// TwinCAT 3 PLC project XtsTransport
// Title: XTS Transport
// Author: HAUD
// ProjectVersion: 4.02.16
// Description: . XTS_TRANSPORT_LAYER by Daniel Hauer
// ProgramVersion: 3.1.4026.22
// libraries:
//   Tc2_EtherCAT, * (Beckhoff Automation GmbH)
//   Tc2_Math, * (Beckhoff Automation GmbH)
//   Tc2_MC2, * (Beckhoff Automation GmbH)
//   Tc2_Standard, * (Beckhoff Automation GmbH)
//   Tc2_System, * (Beckhoff Automation GmbH)
//   Tc2_Utilities, * (Beckhoff Automation GmbH)
//   Tc2_XmlDataSrv, * (Beckhoff Automation GmbH)
//   Tc3_McCollisionAvoidance, * (Beckhoff Automation GmbH)
//   Tc3_McCoordinatedMotion, * (Beckhoff Automation GmbH)
//   Tc3_Module, * (Beckhoff Automation GmbH)
//   Tc3_XTS_Utility, * (Beckhoff Automation GmbH)
//   VisuDialogs, * (System)
// project tree:
//   APPLICATION/ GVL_APPLICATION.TcGVL, MAIN_APP.TcPOU
//   APPLICATION/_config/ StationParameterExample.TcPOU
//   APPLICATION/_types/Application/ E_APP_CHECK.TcDUT, E_APP_VARIANT.TcDUT, ST_APP_CTRL.TcDUT, ST_APP_STATE.TcDUT
//   APPLICATION/_types/Collector/ E_PROCESS_CHECK.TcDUT, E_PROCESS_CTRL.TcDUT, E_PROCESS_STATE.TcDUT, fb_ProcessCollector.TcPOU, fb_StationCollector.TcPOU, I_ProcessCollector.TcIO, ST_PROCESS_CTRL.TcDUT, ST_PROCESS_STATE.TcDUT
//   APPLICATION/_types/ fb_ProcessConductor.TcPOU
//   APPLICATION/_types/Instance/ E_INSTANCE.TcDUT, E_INSTANCE_CHECK.TcDUT, E_INSTANCE_CMD.TcDUT, E_INSTANCE_STATE.TcDUT, fb_Instance.TcPOU, ST_INSTANCE_CTRL.TcDUT, ST_INSTANCE_STATE.TcDUT
//   APPLICATION/_types/LinkedList/ E_LIST_CHECK.TcDUT, E_LIST_CTRL.TcDUT, E_LIST_STATE.TcDUT, fb_Process_LinkedList.TcPOU, fb_Process_LinkedListCtrl.TcPOU, I_Process_LinkedList.TcIO, ST_LIST_CTRL.TcDUT, ST_LIST_NODE_DATA.TcDUT, ST_LIST_STATE.TcDUT, ST_PROCESS_DATA.TcDUT, ST_PROCESS_LIST_RESULT.TcDUT
//   / GlobalTextList.TcGTLO, PlcTask.TcTTO
//   MAPPING/ MAPPING_XTS_in.TcPOU, MAPPING_XTS_out.TcPOU
//   MAPPING/_types/ E_MAPPING_CHECK.TcDUT, U_APP_CTRL.TcDUT, U_APP_STATE.TcDUT, U_GEAR_DATA.TcDUT, U_INSTANCE_CTRL.TcDUT, U_INSTANCE_STATE.TcDUT, U_MOVER_CTRL.TcDUT, U_MOVER_INFO.TcDUT, U_MOVER_SELECTOR_CTRL.TcDUT, U_MOVER_SELECTOR_STATE.TcDUT, U_MOVER_STATE.TcDUT, U_MOVE_DATA.TcDUT, U_TICKET_LIST_CTRL.TcDUT, U_TICKET_LIST_DATA_INPUT.TcDUT, U_TICKET_LIST_DATA_OUTPUT.TcDUT, U_TICKET_LIST_STATE.TcDUT, U_XTS_STATION_CTRL.TcDUT, U_XTS_STATION_STATE.TcDUT, U_XTS_TRANSPORT_CTRL.TcDUT, U_XTS_TRANSPORT_STATE.TcDUT
//   _MSG/class/ fb_LocalTime.TcPOU, fb_MessageData.TcPOU, fb_MessageDataCtrl.TcPOU
//   _MSG/ f_MessageSet.TcPOU, GVL_MSG_AXIS.TcGVL, GVL_MSG_XTS.TcGVL, I_MessageData.TcIO
//   _MSG/types/ e_Device.TcDUT, E_MessageType.TcDUT, E_MESSAGE_BATCH.TcDUT (not stored), E_MESSAGE_CHECK.TcDUT, E_MESSAGE_CTRL.TcDUT, E_MESSAGE_FLOW.TcDUT, E_MESSAGE_STATE.TcDUT, e_Subdevice.TcDUT, ST_Message.TcDUT, ST_MESSAGE_CTRL.TcDUT, ST_MESSAGE_STATE.TcDUT (not stored), TL_E_MESSAGETYPE.TcTLO
//   PLC_MOTION/_GVL/ PLC_CONSTANT.TcGVL
//   _types/ E_CHECK_STATE.TcDUT, E_PROGRESS.TcDUT, f_GetProgress.TcPOU, f_GetState.TcPOU, T_PROCESS.TcDUT
//   _XML/Configuration/ fb_Configuration.TcPOU, I_Configuration_Station.TcIO
//   _XML/Configuration/types/ ST_Configuration.TcDUT
//   _XML/ fb_XmlBase.TcPOU (not stored)
//   _XML/PositionOffsets/ fb_MoverPositionOffsetData.TcPOU
//   _XML/PositionOffsets/types/ ST_MOVER_OFFSETS.TcDUT
//   _XML/types/ E_DATA_CHECK.TcDUT (not stored), E_DATA_CTRL.TcDUT (not stored), E_DATA_STATE.TcDUT, fb_XmlRead.TcPOU (not stored), fb_XmlWrite.TcPOU, ST_DATA_CTRL.TcDUT (not stored), ST_DATA_STATE.TcDUT
//   XTS_TRANSPORT/CaGroup/ FB_CaGroup.TcPOU, I_XtsTransport_CaGroup.TcIO
//   XTS_TRANSPORT/CaGroup/types/ E_CA_GROUP_STATE.TcDUT, E_GROUP_CHECK.TcDUT, ST_GROUP_INFO.TcDUT
//   XTS_TRANSPORT/ GVL_XTS.TcGVL, GVL_XTS_CONSTANTS.TcGVL (not stored), GVL_XTS_VERSION.TcGVL, MAIN_XTS.TcPOU
//   XTS_TRANSPORT/Mover/ fb_Mover.TcPOU, fb_MoverCtrl.TcPOU, fb_MoverSelector.TcPOU (not stored), I_XtsTransport_Mover.TcIO
//   XTS_TRANSPORT/Mover/types/ E_MOVER_CHECK.TcDUT (not stored), E_MOVER_CTRL.TcDUT, E_MOVER_SELECTOR.TcDUT (not stored), E_MOVER_STATE.TcDUT, ST_GEAR_DATA.TcDUT, ST_MOVER_CTRL.TcDUT, ST_MOVER_INFO.TcDUT, ST_MOVER_SELECTOR_CTRL.TcDUT (not stored), ST_MOVER_SELECTOR_STATE.TcDUT, ST_MOVER_STATE.TcDUT, ST_MOVE_DATA.TcDUT
//   XTS_TRANSPORT/Xpu/ I_XtsTransport_Xpu.TcIO, fb_Xpu.TcPOU, fb_XpuCtrl.TcPOU
//   XTS_TRANSPORT/XtsStation/ fb_StationGearInPos.TcPOU, fb_StationProcess.TcPOU, I_XtsTransport_Station.TcIO
//   XTS_TRANSPORT/XtsStation/types/ E_STATION_CHECK.TcDUT, E_STATION_CTRL.TcDUT, E_STATION_GEAR_DISTANCE_AXIS.TcDUT, E_STATION_STATE.TcDUT, E_STATION_TYPE.TcDUT, fb_StationBase.TcPOU, fb_Station_LinkedList.TcPOU, I_Station_LinkedList.TcIO, ST_STATION_CTRL.TcDUT, ST_STATION_GEAR_PARAMETER.TcDUT, ST_STATION_LIST_RESULT.TcDUT, ST_STATION_MOVER_DATA.TcDUT, ST_STATION_PARAMETER.TcDUT, ST_STATION_STATE.TcDUT, T_NEST_OFFSET.TcDUT
//   XTS_TRANSPORT/_Visualization/ GROUP_VISU.TcVIS, MOVER_VISU.TcVIS, SELECTOR_VISU.TcVIS, STATION_VISU.TcVIS, Visualization Manager.TcVMO (not stored), XPU_VISU.TcVIS, XTS_TRANSPORT.TcVIS
//   XTS_TRANSPORT/_Visualization/textlists/ TL_E_CTRL_MOVER.TcTLO, TL_E_CTRL_STATION.TcTLO, TL_E_CTRL_TRANSPORT.TcTLO, TL_E_CTRL_XPU.TcTLO, TL_E_MOVER_SELECTOR.TcTLO
//   XTS_TRANSPORT/_Visualization/types/ T_MOVER_SELECTOR.TcVIS (not stored), ST_XPU_STRINGS.TcDUT
//   XTS_TRANSPORT/Xpu/types/ E_XPU_CHECK.TcDUT, E_XPU_CTRL.TcDUT, E_XPU_INIT.TcDUT, E_XPU_STATE.TcDUT, ST_XPU_CTRL.TcDUT, ST_XPU_INFO.TcDUT, ST_XPU_STATE.TcDUT
//   XTS_TRANSPORT/XtsTransportUnit/ fb_TransportUnit.TcPOU
//   XTS_TRANSPORT/XtsTransportUnit/types/ E_XTS_TRANSPORT_CHECK.TcDUT, E_XTS_TRANSPORT_CTRL.TcDUT, E_XTS_TRANSPORT_STATE.TcDUT, ST_XTS_TRANSPORT_CTRL.TcDUT, ST_XTS_TRANSPORT_STATE.TcDUT

CONFIGURATION XtsTransport
    RESOURCE PLC ON TwinCAT3
        TASK PlcTask(INTERVAL := T#2ms, PRIORITY := 15);
        PROGRAM MAPPING_XTS_in WITH PlcTask : MAPPING_XTS_in;
        PROGRAM MAIN_XTS WITH PlcTask : MAIN_XTS;
        PROGRAM MAIN_APP WITH PlcTask : MAIN_APP;
        PROGRAM MAPPING_XTS_out WITH PlcTask : MAPPING_XTS_out;
    END_RESOURCE
END_CONFIGURATION

// ---- APPLICATION/_types/Application/E_APP_CHECK.TcDUT
{attribute 'qualified_only'}
{attribute 'strict'}
{attribute 'to_string'}
TYPE E_APP_CHECK :
(
  NULL,

  POINTER_CTRL_INVALID                := 9000,
  POINTER_STATE_INVALID,
  REFERENCE_INSTANCE_CONTROL_INVALID,
  REFERENCE_INSTANCE_STATE_INVALID,

	POINTER_TRANSPORT_CTRL_INVALID      := 9100,
	POINTER_TRANSPORT_STATE_INVALID     := 9200,
	POINTER_COLLECTOR_ITF_INVALID       := 9300,
  REFERENCE_PROCESS_LIST_ITF_INVALID  := 9400,

  CHECK_DONE := 10000

)UINT;
END_TYPE

// ---- APPLICATION/_types/Application/E_APP_VARIANT.TcDUT
{attribute 'qualified_only'}
{attribute 'strict'}
{attribute 'to_string'}
{info 'E_APP_VARIANT placeholder for application variant; add new members here'}
TYPE E_APP_VARIANT :
(
  VARIANT_INVALID
);
END_TYPE

// ---- APPLICATION/_types/Application/ST_APP_CTRL.TcDUT
TYPE ST_APP_CTRL :
STRUCT
  Cmd       : E_INSTANCE_CMD;
  Variant   : E_APP_VARIANT;
END_STRUCT
END_TYPE

// ---- APPLICATION/_types/Application/ST_APP_STATE.TcDUT
TYPE ST_APP_STATE :
STRUCT
  AppInit             : E_PROGRESS;
  State            : E_INSTANCE_STATE;
END_STRUCT
END_TYPE

// ---- APPLICATION/_types/Collector/E_PROCESS_CHECK.TcDUT
{attribute 'qualified_only'}
{attribute 'strict'}
{attribute 'to_string'}
TYPE E_PROCESS_CHECK :
(
  NULL,
  REFERENCE_CTRL_INVALID,
  REFERENCE_STATE_INVALID,
  REFERENCE_MOVER_INFO_INVALID,
	STATION_FIRST_ZERO,
  STATION_LAST_ZERO,
  STATION_FIRST_MAX,
  STATION_LAST_MAX,
  STATION_COUNT_NEGATIVE, // last station must have higher index than first station, range must also be closed
  STATION_COUNT_TOO_HIGH, // process can only be max (SIZEOF(T_PROCESS)*8)

  CHECK_DONE    := 10000
);
END_TYPE

// ---- APPLICATION/_types/Collector/E_PROCESS_CTRL.TcDUT
{attribute 'qualified_only'}
{attribute 'strict'}
{attribute 'to_string'}
TYPE E_PROCESS_CTRL :
(
  PROCESS_INIT              := 10,
  PROCESS_DISABLE           := 20,
  PROCESS_ENABLE            := 30,
  PROCESS_STATIONS_INFEED,

  PROCESS_STATIONS_ENTER    := 40,
  PROCESS_STATIONS_SEND,

  PROCESS_START             := 60,
  PROCESS_DONE              := 70,
  PROCESS_STATIONS_OUTFEED  := 80
);
END_TYPE

// ---- APPLICATION/_types/Collector/E_PROCESS_STATE.TcDUT
{attribute 'qualified_only'}
{attribute 'strict'}
{attribute 'to_string'}
TYPE E_PROCESS_STATE :
(
  PROCESS_INVALID,
  PROCESS_NO_INIT,
  PROCESS_INIT              := 10,
  PROCESS_DISABLE           := 20,
  PROCESS_ENABLE            := 30,
  PROCESS_STATIONS_INFEED   := 40,
  PROCESS_STATIONS_NEST,

  PROCESS_START             := 60,
  PROCESS_DONE              := 70,
  PROCESS_STATIONS_OUTFEED  := 80
);
END_TYPE

// ---- APPLICATION/_types/Collector/ST_PROCESS_CTRL.TcDUT
{attribute 'pack_mode' := '2'}
TYPE ST_PROCESS_CTRL :
STRUCT
  Cmd               : E_PROCESS_CTRL;
  ProcessTarget     : UINT;
  ActivateStation   : T_PROCESS;  // every bit is a XtsStation
  NestMask          : BYTE;       // every bit is a PosStop in a XtsStation, one mask for all XtsStations, copied to every XtsStation control in process
END_STRUCT
END_TYPE

// ---- APPLICATION/_types/Collector/ST_PROCESS_STATE.TcDUT
{attribute 'pack_mode' := '2'}
TYPE ST_PROCESS_STATE :
STRUCT
  State           : E_PROCESS_STATE;
  Result          : E_PROGRESS;
  Check           : E_PROCESS_CHECK;
END_STRUCT
END_TYPE

// ---- APPLICATION/_types/Instance/E_INSTANCE.TcDUT
{attribute 'qualified_only'}
{attribute 'strict'}
{attribute 'to_string'}
{info 'E_INSTANCE placeholder for process identification; add new members here'}
TYPE E_INSTANCE : // placeholder for process identification; add new members here
(
	INSTANCE_NULL,
  // list your process instances here
  INSTANCE_EXAMPLE,
  INSTANCE_MAX
)UINT;
END_TYPE

// ---- APPLICATION/_types/Instance/E_INSTANCE_CHECK.TcDUT
{attribute 'qualified_only'}
{attribute 'strict'}
{attribute 'to_string'}
TYPE E_INSTANCE_CHECK :
(
  NULL,

	POINTER_COLLECTOR_ITF_INVALID := 9000,
  INVALID_INSTANCE_CONTROL_REFERENCE,
  INVALID_INSTANCE_STATE_REFERENCE,
  PROCESS_ID_ZERO := 9100,
  PROCESS_ID_MAX  := 9200,
  PROCESS_ID_NOTEQUAL_COLLECTOR_ID := 9300,
  PROCESS_LIST_ITF_INDEX_INVALID := 9400,

  CHECK_DONE := 10000
)UINT;
END_TYPE

// ---- APPLICATION/_types/Instance/E_INSTANCE_CMD.TcDUT
{attribute 'qualified_only'}
{attribute 'to_string'}
{attribute 'strict'}
TYPE E_INSTANCE_CMD : // instructions for fb_Instance executions
(
	NULL,
  INIT,
  DISABLE,
  ENABLE,
  WORK,
  PROCEED := 100,
  FINISH,
  CLEAR
)UINT;
END_TYPE

// ---- APPLICATION/_types/Instance/E_INSTANCE_STATE.TcDUT
{attribute 'qualified_only'}
//{attribute 'strict'}
{attribute 'to_string'}
TYPE E_INSTANCE_STATE :
(
  NULL,
	INVALID,
  INIT,
  DISABLED,
  DETECTION,
  ENABLED,
  WORKING,
  PROCEEDING,
  FINISH,
  CLEARED
)UINT;
END_TYPE

// ---- APPLICATION/_types/Instance/ST_INSTANCE_CTRL.TcDUT
TYPE ST_INSTANCE_CTRL :
STRUCT
  Cmd     : E_INSTANCE_CMD;
END_STRUCT
END_TYPE

// ---- APPLICATION/_types/Instance/ST_INSTANCE_STATE.TcDUT
{attribute 'pack_mode' := '2'}
TYPE ST_INSTANCE_STATE :
STRUCT
  State             : E_INSTANCE_STATE;
  Progress          : E_PROGRESS;

  QueueProcessCount : UINT; // sum of all queues in process
  StationCount      : UINT;
END_STRUCT
END_TYPE

// ---- APPLICATION/_types/LinkedList/E_LIST_CHECK.TcDUT
{attribute 'qualified_only'}
{attribute 'strict'}
{attribute 'to_string'}
TYPE E_LIST_CHECK :
(
	CHECK_NULL,
  CHECK_INVALID_REF_CTRL,
  CHECK_INVALID_REF_STATE,
  CHECK_INVALID_REF_DATA_INPUT,
  CHECK_INVALID_REF_DATA_OUTPUT,

  CHECK_DONE              := 10000
);
END_TYPE

// ---- APPLICATION/_types/LinkedList/E_LIST_CTRL.TcDUT
{attribute 'qualified_only'}
{attribute 'strict'}
{attribute 'to_string'}
TYPE E_LIST_CTRL :
(
  LIST_CTRL_INVALID,
	LIST_CTRL_NULL,
  LIST_CTRL_INIT      := 10,
  LIST_CTRL_GET_HEAD  := 20,
  LIST_CTRL_GET_TAIL  := 30,
  LIST_CTRL_ADD_HEAD  := 40,
  LIST_CTRL_ADD_TAIL  := 50,
  LIST_CTRL_DEL_HEAD  := 60,
  LIST_CTRL_DEL_TAIL  := 70
)UINT;
END_TYPE

// ---- APPLICATION/_types/LinkedList/E_LIST_STATE.TcDUT
{attribute 'qualified_only'}
//{attribute 'strict'}
{attribute 'to_string'}
TYPE E_LIST_STATE :
(
  LIST_STATE_INVALID,
	LIST_STATE_NULL,
  LIST_STATE_INIT      := 10,
  LIST_STATE_GET_HEAD  := 20,
  LIST_STATE_GET_TAIL  := 30,
  LIST_STATE_ADD_HEAD  := 40,
  LIST_STATE_ADD_TAIL  := 50,
  LIST_STATE_DEL_HEAD  := 60,
  LIST_STATE_DEL_TAIL  := 70
)UINT;
END_TYPE

// ---- APPLICATION/_types/LinkedList/ST_LIST_CTRL.TcDUT
TYPE ST_LIST_CTRL :
STRUCT
  Cmd         : E_LIST_CTRL;
END_STRUCT
END_TYPE

// ---- APPLICATION/_types/LinkedList/ST_LIST_NODE_DATA.TcDUT
{attribute 'pack_mode' := '2'}
TYPE ST_LIST_NODE_DATA :
STRUCT
  ProcessData     : ST_PROCESS_DATA;  // target data
END_STRUCT
END_TYPE

// ---- APPLICATION/_types/LinkedList/ST_LIST_STATE.TcDUT
{attribute 'pack_mode' := '2'}
TYPE ST_LIST_STATE :
STRUCT
  Init        : E_PROGRESS;
  State       : E_LIST_STATE;

  Free        : UDINT;
  Count       : UDINT;
END_STRUCT
END_TYPE

// ---- APPLICATION/_types/LinkedList/ST_PROCESS_DATA.TcDUT
TYPE ST_PROCESS_DATA :
STRUCT
  nProcessId          : e_instance; // target process
  {attribute 'displaymode':='bin'}
  wTarget             : T_PROCESS;  // where and how many stations are to be used in process
END_STRUCT
END_TYPE

// ---- APPLICATION/_types/LinkedList/ST_PROCESS_LIST_RESULT.TcDUT
TYPE ST_PROCESS_LIST_RESULT :
STRUCT
  wState    : WORD;   // wState == 0 --> all ok
  nIndex    : ULINT;
  stData    : ST_PROCESS_DATA;  // copy of list entry
END_STRUCT
END_TYPE

// ---- MAPPING/_types/E_MAPPING_CHECK.TcDUT
{attribute 'qualified_only'}
{attribute 'strict'}
{attribute 'to_string'}
TYPE E_MAPPING_CHECK :
(
  NULL,
  MAPPING_NOT_ACTIVE,
  
  MOVER_CTRL_SIZE_MISSMATCH   := 9000,
  MOVER_STATE_SIZE_MISSMATCH,
  MOVER_INFO_SIZE_MISSMATCH,
  MOVE_DATA_SIZE_MISSMATCH,
  GEAR_DSTS_SIZE_MISSMATCH,

  TRANSPORT_CTRL_MISSMATCH,
  TRANSPORT_STATE_MISSMATCH,


  STATION_CTRL_SIZE_MISSMATCH,
  STATION_STATE_SIZE_MISSMATCH,

  APP_CTRL_SIZE_MISSMATCH     := 9100,
  APP_STATE_SIZE_MISSMATCH,

  INSTANCE_CTRL_SIZE_MISSMATCH,
  INSTANCE_STATE_SIZE_MISSMATCH,


  CHECK_DONE                  := 10_000

  
);
END_TYPE

// ---- MAPPING/_types/U_APP_CTRL.TcDUT
TYPE U_APP_CTRL :
UNION
  stCtrl              : ST_APP_CTRL;
  byCtrl    AT %I*    : ARRAY[1..SIZEOF(ST_APP_CTRL)] OF BYTE;
END_UNION
END_TYPE

// ---- MAPPING/_types/U_APP_STATE.TcDUT
TYPE U_APP_STATE :
UNION
  stState             : ST_APP_STATE;
  byState   AT %Q*    : ARRAY[1..SIZEOF(ST_APP_STATE)] OF BYTE;
END_UNION
END_TYPE

// ---- MAPPING/_types/U_GEAR_DATA.TcDUT
TYPE U_GEAR_DATA :
UNION
  stData              : ARRAY[1..MAX_MOVER] OF ST_GEAR_DATA;

  byData    AT %I*    : ARRAY[1..MAX_MOVER] OF
                        ARRAY[1..SIZEOF(ST_GEAR_DATA)] OF BYTE;
END_UNION
END_TYPE

// ---- MAPPING/_types/U_INSTANCE_CTRL.TcDUT
TYPE U_INSTANCE_CTRL :
UNION
  stCtrl              : ARRAY[1..MAX_PROCESS] OF ST_INSTANCE_CTRL;
  byCtrl    AT %I*    : ARRAY[1..MAX_PROCESS] OF
                        ARRAY[1..SIZEOF(ST_INSTANCE_CTRL)] OF BYTE;
END_UNION
END_TYPE

// ---- MAPPING/_types/U_INSTANCE_STATE.TcDUT
TYPE U_INSTANCE_STATE :
UNION
  stState             : ARRAY[1..MAX_PROCESS] OF ST_INSTANCE_STATE;
  byState   AT %Q*    : ARRAY[1..MAX_PROCESS] OF
                        ARRAY[1..SIZEOF(ST_INSTANCE_STATE)] OF BYTE;
END_UNION
END_TYPE

// ---- MAPPING/_types/U_MOVER_CTRL.TcDUT
TYPE U_MOVER_CTRL :
UNION
  stCtrl              : ARRAY[1..MAX_MOVER] OF ST_MOVER_CTRL;

  byCtrl    AT %I*    : ARRAY[1..MAX_MOVER] OF
                        ARRAY[1..SIZEOF(ST_MOVER_CTRL)] OF BYTE;
END_UNION
END_TYPE

// ---- MAPPING/_types/U_MOVER_INFO.TcDUT
TYPE U_MOVER_INFO :
UNION
  stInfo              : ARRAY[1..MAX_MOVER] OF ST_MOVER_INFO;

  byInfo    AT %Q*    : ARRAY[1..MAX_MOVER] OF
                        ARRAY[1..SIZEOF(ST_MOVER_INFO)] OF BYTE;
END_UNION
END_TYPE

// ---- MAPPING/_types/U_MOVER_SELECTOR_CTRL.TcDUT
TYPE U_MOVER_SELECTOR_CTRL :
UNION
  stCtrl              : ST_MOVER_SELECTOR_CTRL;

  byCtrl    AT %I*    : ARRAY[1..SIZEOF(ST_MOVER_SELECTOR_CTRL)] OF BYTE;

END_UNION
END_TYPE

// ---- MAPPING/_types/U_MOVER_SELECTOR_STATE.TcDUT
TYPE U_MOVER_SELECTOR_STATE :
UNION
  stState             : ST_MOVER_SELECTOR_STATE;

  byState   AT %Q*    : ARRAY[1..SIZEOF(ST_MOVER_SELECTOR_STATE)] OF BYTE;
END_UNION
END_TYPE

// ---- MAPPING/_types/U_MOVER_STATE.TcDUT
TYPE U_MOVER_STATE :
UNION
  stState             : ARRAY[1..MAX_MOVER] OF ST_MOVER_STATE;

  byState   AT %Q*    : ARRAY[1..MAX_MOVER] OF
                        ARRAY[1..SIZEOF(ST_MOVER_STATE)] OF BYTE;
END_UNION
END_TYPE

// ---- MAPPING/_types/U_MOVE_DATA.TcDUT
TYPE U_MOVE_DATA :
UNION
  stData              : ARRAY[1..MAX_MOVER] OF ST_MOVE_DATA;

  byData    AT %I*    : ARRAY[1..MAX_MOVER] OF
                        ARRAY[1..SIZEOF(ST_MOVE_DATA)] OF BYTE;
END_UNION
END_TYPE

// ---- MAPPING/_types/U_TICKET_LIST_CTRL.TcDUT
TYPE U_TICKET_LIST_CTRL :
UNION
  stCtrl              : ST_LIST_CTRL;
  byCtrl    AT %I*    : ARRAY[1..SIZEOF(ST_LIST_CTRL)] OF BYTE;
END_UNION
END_TYPE

// ---- MAPPING/_types/U_TICKET_LIST_DATA_INPUT.TcDUT
TYPE U_TICKET_LIST_DATA_INPUT :
UNION
  stData              : ST_LIST_NODE_DATA;
  byData   AT %I*     : ARRAY[1..SIZEOF(ST_LIST_NODE_DATA)] OF BYTE;
END_UNION
END_TYPE

// ---- MAPPING/_types/U_TICKET_LIST_DATA_OUTPUT.TcDUT
TYPE U_TICKET_LIST_DATA_OUTPUT :
UNION
  stData              : ST_LIST_NODE_DATA;
  byData   AT %Q*     : ARRAY[1..SIZEOF(ST_LIST_NODE_DATA)] OF BYTE;
END_UNION
END_TYPE

// ---- MAPPING/_types/U_TICKET_LIST_STATE.TcDUT
TYPE U_TICKET_LIST_STATE :
UNION
  stState             : ST_LIST_STATE;
  byState   AT %Q*    : ARRAY[1..SIZEOF(ST_LIST_STATE)] OF BYTE;
END_UNION
END_TYPE

// ---- MAPPING/_types/U_XTS_STATION_CTRL.TcDUT
TYPE U_XTS_STATION_CTRL :
UNION
  stCtrl              : ARRAY[1..MAX_STATION] OF ST_STATION_CTRL;

  byCtrl    AT %I*    : ARRAY[1..MAX_STATION] OF
                        ARRAY[1..SIZEOF(ST_STATION_CTRL)] OF BYTE;
END_UNION
END_TYPE

// ---- MAPPING/_types/U_XTS_STATION_STATE.TcDUT
TYPE U_XTS_STATION_STATE :
UNION
  stState             : ARRAY[1..MAX_STATION] OF ST_STATION_STATE;

  byState   AT %Q*    : ARRAY[1..MAX_STATION] OF
                        ARRAY[1..SIZEOF(ST_STATION_STATE)] OF BYTE;
END_UNION
END_TYPE

// ---- MAPPING/_types/U_XTS_TRANSPORT_CTRL.TcDUT
{attribute 'pack_mode' := '2'}
TYPE U_XTS_TRANSPORT_CTRL :
UNION
  stCtrl              : ST_XTS_TRANSPORT_CTRL;
  byCtrl    AT %I*    : ARRAY[1..SIZEOF(ST_XTS_TRANSPORT_CTRL)] OF BYTE;
END_UNION
END_TYPE

// ---- MAPPING/_types/U_XTS_TRANSPORT_STATE.TcDUT
{attribute 'pack_mode' := '2'}
TYPE U_XTS_TRANSPORT_STATE :
UNION
  stState             : ST_XTS_TRANSPORT_STATE;
  byState   AT %Q*    : ARRAY[1..SIZEOF(ST_XTS_TRANSPORT_STATE)] OF BYTE;
END_UNION
END_TYPE

// ---- _MSG/types/e_Device.TcDUT
{attribute 'to_string'}
TYPE e_Device :
(
  Device_Null,                  // NULL               - not to be used
  Device_Main,                  // MAIN(PRG)          - reserved for MAIN(PRG)
  Device_MainAxis,              // MAIN_AXIS(PRG)     - reserved for MAIN_AXIS(PRG)
  Device_Nci,                   // NCI(PRG)           - reserved for NCI(PRG)
  Device_Cam,                   // CAM(PRG            - reserved for CAM(PRG)
  Device_Functions,             // FUNCTIONS(PRG)     - reserved for FUNCTIONS(PRG)
  Device_FlyingSaw,             // FLYING_SAW(PRG)    - reserved for FLYING_SAW(PRG)
  Device_MainApplication,       // MAIN_APP(PRG)      - reserved for MAIN_APP(PRG)

  Device_MoverSelector,         // single mover interface for xts applications
  Device_ParameterSelector,     // fb_ParameterSelector can only exist once in a project.
  Device_Configuration,         // fb_Configuration can handle multiple files therefore only one instance is required
  Device_XmlData,               // generic XML Data (e.g. persistent data)
  Device_Utilities,             // service calls to anyone you may want to talk to, the main intent is to get XPU and TcXtsIo data to the application side

  General           :=  1000,
  CaGroup           :=  2000,
  Xpu               :=  3000,
  XpuCtrl           :=  4000,
  Mover             :=  5000,
  MoverCtrl         :=  6000,
  XtsTransportUnit  :=  7000,
  XfcTriggerBox     :=  8000,
  XfcTouchProbe     :=  9000,
  XtsStation        := 10000,

  Camming           := 11000,
  NciChannel        := 12000,
  NciChannelCtrl    := 13000,
  Axis              := 14000,
  XfcAxis           := 15000,

  // txt file logging LOG_FILE_METRICS
  MetricsXts        := 16000,   //entries from xts Metrics are written into dedicated txt file (see f_MessageSet, here's the diverter)
  MetricsAxis       := 17000,   //entries from PLC_MOTION Metrics are written into dedicated txt file

  // txt file logging LOG_FILE_APP
  Process           := 20000,   // entries from process are written into dedicated txt file.
  ProcessListCtrl   := 21000,
  TicketListCtrl    := 22000,

  Application       := 30000,   // entries from application are written into dedicated txt file.


  // txt file logging LOG_FILE_PRODUCT - this is for you to use
  DataProduct       := 40000
)UDINT;
END_TYPE

// ---- _MSG/types/E_MessageType.TcDUT
{attribute 'strict'}
{attribute 'to_string'}
TYPE E_MessageType :
(
  //-----------------------------------------------------
  //-----------------------------------------------------
  //  message system:
  //  - errors are always calling f_MessageSet()
  //  - errors are always entered into its list
  //
  //  - message severity is set by this enum (like everywhere else)
  //
  //  - message frequency is set by this enum
  //    - IF you get above 50 stations, 
  //      writing to the file system takes time:
  //
  //    Batch: switching on metrics (> Empty) must not add cpu load, 
  //      --> so do not clutter here
  //
  //    Info:  regular flow of information (>Error / >Warning) 
  //           must not add significant cpu load, 
  //      --> so do not clutter here
  //
  //    Verbose and above:
  //    --> for small systems (< 96 mover, < 50 stations) 
  //        you may switch it on for everybody, 
  //        files get big quickly ;-)
  //
  //    --> switch on during test phase for a handful of stations
  //
  //    --> high detail logging always and for everybody
  //    --> we need somebody who transfers data more quickly
  //      --> I can offer a .NET(C#) ADS tool which collects the list.
  //          .NET application then pushes to database
  //-----------------------------------------------------
  //-----------------------------------------------------
  eMessageEmpty,    // he who is without bounds may speak
  eMessageBatch,    // he who counts words, counts numbers (Batch started, Next in Batch, Batch done)
  eMessageError,    // mine, your(')s, anybody's, let the numbers tell you
  eMessageWarning,  // I told you so
  eMessageInfo,     // A long time ago in a galaxy far, far away...
  eMessageVerbose,  // He talks a lot, doesn't he?; Yeah! He's very knowledgeable.
  eMessageSentient  // Keep them out of bright light, Don't get them wet, do not feed them after midnight!! No matter how much they beg!!
)DINT;
END_TYPE

// ---- _MSG/types/E_MESSAGE_CHECK.TcDUT
{attribute 'qualified_only'}
{attribute 'strict'}
{attribute 'to_string'}
TYPE E_MESSAGE_CHECK :
(
  NULL,
  // 9000 --> here comes your error
  POINTER_INVALID             := 9000,
  POINTER_TIME_INVALID,
  POINTER_LIST_INVALID,
  POINTER_MSG_IDX_INVALID,
  POINTER_ERR_IDX_INVALID,
  POINTER_ROOT_FILE_INVALID,
  POINTER_ROOT_DIR_INVALID,
  POINTER_CTRL_INVALID,
  POINTER_STATE_INVALID,

  // 10000 --> here comes your man
  CHECK_DONE                        := 10000
)UINT;
END_TYPE

// ---- _MSG/types/E_MESSAGE_CTRL.TcDUT
{attribute 'qualified_only'}
{attribute 'strict'}
{attribute 'to_string'}
TYPE E_MESSAGE_CTRL :
(
	MSG_CTRL_NULL,
	MSG_CTRL_INIT   := 10,
  MSG_CTRL_IDLE   := 30,
  MSG_CTRL_WRITE  := 50
)UINT;
END_TYPE

// ---- _MSG/types/E_MESSAGE_FLOW.TcDUT
{attribute 'qualified_only'}
{attribute 'strict'}
{attribute 'to_string'}
TYPE E_MESSAGE_FLOW :
(
  MSG_FLOW_INIT,
  MSG_FLOW_ROOT                 := 10,
  MSG_FLOW_ROOT_CREATE,
  MSG_FLOW_ROOT_CREATE_BUSY,
  MSG_FLOW_FOLDER,
  MSG_FLOW_FOLDER_CREATE,
  MSG_FLOW_FOLDER_CREATE_BUSY,
  MSG_FLOW_FILE_CREATE_DONE,
  MSG_FLOW_LINE_START           := 100,
  MSG_FLOW_LINE_BUILD,
  MSG_FLOW_LINE_CHECK,
  MSG_FLOW_WRITE_FILE_BUSY      := 200,
  MSG_FLOW_WRITE_FILE_END,
  MSG_FLOW_WRITE_FILE_DONE      := 1000
)UINT;
END_TYPE

// ---- _MSG/types/E_MESSAGE_STATE.TcDUT
{attribute 'qualified_only'}
//{attribute 'strict'}
{attribute 'to_string'}
TYPE E_MESSAGE_STATE :
(
	MSG_STATE_NULL,
  MSG_STATE_INIT    := 10,
  MSG_STATE_IDLE    := 30,
  MSG_STATE_WRITE   := 50
)UINT;
END_TYPE

// ---- _MSG/types/e_Subdevice.TcDUT
{attribute 'strict'}
{attribute 'to_string'}
TYPE e_Subdevice :
(
  // sub device for message system
  General                 :=  0,
  MainInit,
  // Motion Control FB Instances
  fbPower,
  fbReset,
  fbResetSercos,
  fbHalt,
  fbStop,                 // 5
  fbHome,
  fbJog,
  fbMoveVelocity1,
  fbMoveVelocity2,
  fbMoveAbsolute1,        // 10
  fbMoveAbsolute2,
  fbMoveEndless,
  fbMovePtP,
  fbMoveVelo,
  fbSendToPos,

  // CA CollisionAvoidance FB instances
  // CA group fb instances
  fbCaGroup             := 30,
  fbMoveToPosCa,
  fbSendToAbsPosCa,
  fbSendToModuloPosCa,
  fbGearInPosCa,
  fbGroupAddAxis,
  fbGroupRemoveAxis,
  fbGroupDisable,
  fbGroupEnable,
  fbGroupErrorRead,
  fbGroupStatusRead,
  fbGroupReset,
  fbGroupStop,
  fbHaltCa,

  fbGearIn                := 50,
  fbGearOut,
  fbGearInMultiMaster,

  fbCamOutV2              := 80,
  fbCamInV2,
  fbCamScalingV2,
  fbCamInfoV2,
  fbReadMotionFunction,
  fbReadMotionFunctionPoint,
  fbReadMotionFunctionValues,
  fbWriteMotionFunction,
  fbWriteMotionFunctionPoint,
  fbSetOnlineChangeMode,

  fbReadParameter         := 100,
  fbReadBoolParameter,
  fbWriteParameter,
  fbWriteBoolParameter,
  fbWriteParameterPersistent,
  fbXmlRead,
  fbXmlWrite,
  fbCreateFolder,

  fbBuildGroup            := 200,
  fbClearGroup,
  fbLoadProg,
  fbResetItp,
  fbStartStopItp,
  fbEStopItp,             // 205
  fbStepOnAfterEStopItp,
  fbConfirmHskItp,
  fbDelDtgItp,
  fbNciFeedTablePreparation,
  fbNciFeedTable,         // 210
  fbReadLine,
  fbItpReadRParams,
  fbItpWriteRParams,
  Get_ItpState,
  Get_Error,              // 215


  XfcPositionAtTime       := 300,
  XfcTimeOfPosition,
  XfcTimeToPosition,
  XfcTimeToModuloPosition,
  XfcRecordedPosition,
  XfcTouchProbe,          // 305
  XfcTouchProbeEL1258,
  XfcTouchProbeOptions,
  XfcTriggerRef,
  XfcTriggerRef_MT,
  XfcEl1258Interface_MT,  // 310
  XfcRecordedPosition_MT,
  XfcTriggerOut,
  XfcTriggerStart,
  XfcSwitchOn_2252,
  XfcSwitchOff_2252,      // 315
  XfcInit,
  XfcLatchPosition,
  XfcWaitForPosition,

  AxisMode              := 1000,
  AxisControl,
  AxisStartUp,
  AxisCycle,
  AxisIdle,

  NciControl            := 2000,
  NciStartUp,
  NciCycle,
  NciIdle,

  FlyingSawControl      := 2100,
  FlyingSawStartUp,

  StationLinkedList     := 3000,
  StationInitList,
  StationAddHead,
  StationAddTail,
  StationGetHead,
  StationRemoveHeadValue,
  StationGearInDistanceToSync,
  StationGearInSyncStart,
  StationGearInSyncMove,
  StationGearInSyncEnd,
  StationCalcInfeedPosition,

  StationControl        := 4000,
  StationState, 

  Xpu_fbEnvironment     := 5000,
  Xpu_fbProcessingUnit,
  Xpu_fbXpuPart,
  Xpu_fbXpuTrack,
  Xpu_fbMc2CaGroup,
  Xpu_fbParameterSet,
  Xpu_fbNctController,

  Xpu_fbPartModules     := 5500,

  Xpu_fbMoverXpu        := 6000,

  Xpu_fbNctBaseUnit     := 6500,

  TransportUnit_General := 7000,
  TransportUnit_Restart := 7010,
  TransportUnit_Start,
  TransportUnit_XpuInit,
  TransportUnit_StationClearOutfeed,
  TransportUnit_GroupEnable,
  TransportUnit_GroupClear,
  TransportUnit_GroupBuild,
  TransportUnit_GroupStop,
  TransportUnit_MoverEnableAll,
  TransportUnit_MoverDisableAll,


  CamControl            := 8000,
  CamStartUp,
  CamCycle,

  Process_StationCollector    := 11000,
  Process_ProcessCollector    := 11100,
  Process_ProcessCollector_Init,
  Process_ProcessCollector_Cycle,
  Process_ProcessCollector_Control,

  Process_LinkedList_GetHead,
  Process_LinkedList_RemoveHead,
  Process_LinkedList_AddTail,
  Process_LinkedList_CheckData,
  Process_StationQueue_Check,

  Process_LinkedList_Com              := 11200,
  Process_LinkedList_Com_Init,
  Process_LinkedList_Com_Cmd,
  Process_LinkedList_Com_AddHead,
  Process_LinkedList_Com_AddTail,
  Process_LinkedList_Com_DelHead,
  Process_LinkedList_Com_DelTail,
  Process_LinkedList_Com_GetHead,
  Process_LinkedList_Com_GetTail,


  Instance_Command              := 12000,
  Instance_ProcessConductor,
  Instance_BufferInfeed,
  Instance_Infeed,
  Instance_BufferOutfeed,
  Instance_Outfeed,
  Instance_Sender_Buffer,

  Ticket_LinkedList_Ctrl        := 12100,
  Ticket_LinkedList_Com_Init,
  Ticket_LinkedList_Com_Cmd,
  Ticket_LinkedList_Com_AddHead,
  Ticket_LinkedList_Com_AddTail,
  Ticket_LinkedList_Com_DelHead,
  Ticket_LinkedList_Com_DelTail,
  Ticket_LinkedList_Com_GetHead,
  Ticket_LinkedList_Com_GetTail,
  

  Application                 := 13000,
  Application_Check,
  Application_Clear,
  Application_Cmd,
  Application_Disable,
  Application_Enable,
  Application_Finish,
  Application_Init,
  Application_Proceed,
  Application_Work,

  Utilities                   := 13100,
  Utilities_GetStationOnModule,
  Utilities_SetGlobalConstraints

)DINT;
END_TYPE

// ---- _MSG/types/ST_Message.TcDUT
TYPE ST_Message :
STRUCT
  eType         : e_MessageType;
  eDevice       : e_Device;
  eSubdevice    : e_SubDevice;
  {attribute 'displaymode':='hex'}
  iErrorNumber  : LINT;
  tTime         : STRING(24);
  sText         : STRING(127);
END_STRUCT
END_TYPE

// ---- _MSG/types/ST_MESSAGE_CTRL.TcDUT
TYPE ST_MESSAGE_CTRL :
STRUCT
  Cmd         : E_MESSAGE_CTRL;
END_STRUCT
END_TYPE

// ---- _types/E_CHECK_STATE.TcDUT
{attribute 'qualified_only'}
{attribute 'strict'}
{attribute 'to_string'}
TYPE E_CHECK_STATE :
(
  CHECK_INIT,
  AXIS_INDEX_OUT_OF_RANGE         :=  10,

	AXIS_REF_POINTER_INVALID        := 100,
  AXIS_CTRL_POINTER_INVALID,
  AXIS_STATE_POINTER_INVALID,
  AXIS_INFO_POINTER_INVALID,
  AXIS_DATA_POINTER_INVALID,
  AXIS_NC_PARAMETER_POINTER_INVALID,
  AXIS_HOME_PARAMETER_POINTER_INVALID,
  AXIS_GEAR_IN_PARAMETER_POINTER_INVALID,
  AXIS_GEAR_IN_MULTIMASTER_POINTER_INVALID,
  AXIS_MOTION_OPTIONS_POINTER_INVALID,

  NCI_NOT_ACTIVATED               := 200,
  NCI_CHANNEL_REF_POINTER_INVALID,
  NCI_AXIS_CONFIG_POINTER_INVALID,
  NCI_MCS_AXIS_POINTER_INVALID,
  NCI_AUX_AXIS_POINTER_INVALID,
  NCI_CTRL_POINTER_INVALID,
  NCI_STATE_POINTER_INVALID,
  NCI_R_PARAMETER_READ_POINTER_INVALID,
  NCI_R_PARAMETER_wRITE_POINTER_INVALID,
  NCI_M_FUNC_POINTER_INVALID,

  CAM_NOT_ACTIVATED               := 300,
  CAM_SLAVE_AXIS_REF_INVALID,
  CAM_SLAVE_ITF_MC_AXIS_INVALID,
  CAM_MASTER_AXIS_REF_INVALID,
  CAM_MOTION_FUNCTION_POINTER_INVALID,
  CAM_MOTION_FUNCTION_POINT_POINTER_INVALID,
  AXIS_LIMIT_SWITCHES_POINTER_INVALID,

  FLYING_SAW_NOT_ACTIVATED        := 400,
  FLYING_SLAVE_ITF_MC_AXIS_INVALID,
  FLYING_MASTER_AXIS_REF_INVALID,
  FLYING_FLY_DATA_POINTER_INVALID,
  FLYING_MOVE_DATA_POINTER_INVALID,
  FLYING_OPTIONS_POINTER_INVALID,
  FLYING_OPTIONS_SYNCMODE_SIZE_NOT_EQUAL,

  PARAMETER_SELECTOR              := 500,
  PARAMETER_SELECTOR_CTRL_REF_INVALID,
  PARAMETER_SELECTOR_STATE_REF_INVALID,
  PARAMETER_SELECTOR_AXIS_ITF_INVALID,


  CHECK_DONE                      := 10000
  
)UINT;
END_TYPE

// ---- _types/E_PROGRESS.TcDUT
{attribute 'qualified_only'}
//{attribute 'strict'}
{attribute 'to_string'}
TYPE E_PROGRESS :
(
  // progress has 2 use cases
  // 1. as offset to cyclic interface's state 
  //    for the requested command/function
  //    e.g. State := <Enum equivalent to eCmd> + E_PROGRESS
  //
  // 2. as state feedback (result) from (any) method
  PROGRESS_INVALID,
  PROGRESS_NOT_EXIST      :=   100,
  PROGRESS_INIT           :=  1000,
  PROGRESS_BUSY           :=  2000,
  PROGRESS_PREPARE        :=  3000,
  PROGRESS_STARTUP        :=  4000,
  PROGRESS_CHECK          :=  5000,
  PROGRESS_OCCUPIED       :=  6000,
  PROGRESS_WORKING        :=  7000,
  PROGRESS_STILL_WORKING  :=  8000,
  PROGRESS_ERROR          :=  9000,
  PROGRESS_DONE           := 10000
)UINT;
END_TYPE

// ---- _types/T_PROCESS.TcDUT
TYPE T_PROCESS : DWORD; END_TYPE

// ---- _XML/Configuration/types/ST_Configuration.TcDUT
TYPE ST_Configuration :
STRUCT
  XtsStationParameter  : ARRAY[1..MAX_STATION] OF ST_STATION_PARAMETER;
END_STRUCT
END_TYPE

// ---- _XML/PositionOffsets/types/ST_MOVER_OFFSETS.TcDUT
TYPE ST_MOVER_OFFSETS :
STRUCT
  // static position offsets in stations
  PositionOffset      : ARRAY[1..MAX_STATION] OF T_NEST_OFFSET; // added to PosStop[] in XtsStation
END_STRUCT
END_TYPE

// ---- _XML/types/E_DATA_STATE.TcDUT
{attribute 'qualified_only'}
{attribute 'to_string'}
TYPE E_DATA_STATE :
(
	NULL,
  NO_EXIST,
  INIT        := 10,
  READ        := 20,
  WRITE       := 30
)UINT;
END_TYPE

// ---- _XML/types/ST_DATA_STATE.TcDUT
{attribute 'pack_mode' := '2'}
TYPE ST_DATA_STATE :
STRUCT
  State       : E_DATA_STATE;
  Init        : E_PROGRESS;
END_STRUCT
END_TYPE

// ---- XTS_TRANSPORT/CaGroup/types/E_CA_GROUP_STATE.TcDUT
// {attribute 'qualified_only'}
// {attribute 'strict'}
{attribute 'to_string'}
TYPE E_CA_GROUP_STATE :
(
  // replicated from MC_GROUP_STATE for getting to_string() functionality
	mcGroupStateInvalid   :=0, 
  mcGroupStateDisabled  :=1, 
  mcGroupStateStandby   :=2, 
  mcGroupStateMoving    :=3, 
  mcGroupStateStopping  :=4, 
  mcGroupStateErrorStop :=5, 
  mcGroupStateHoming    :=6, 
  mcGroupStateNotReady  :=7, 
  mcGroupStateSuspended :=8 
)UINT;
END_TYPE

// ---- XTS_TRANSPORT/CaGroup/types/E_GROUP_CHECK.TcDUT
{attribute 'qualified_only'}
{attribute 'to_string'}
TYPE E_GROUP_CHECK :
(
  NULL,
  REFERENCE_GROUP_REF_INVALID := 9000,
  REFERENCE_AXIS_REF_INVALID,
  REFERENCE_CTRL_INVALID,
  REFERENCE_STATE_INVALID,
  REFERENCE_MOVER_ITF_INVALID,
  REFERENCE_XPU_INFO_INVALID,

  CHECK_DONE              := 10000
)UINT;
END_TYPE

// ---- XTS_TRANSPORT/CaGroup/types/ST_GROUP_INFO.TcDUT
TYPE ST_GROUP_INFO :
STRUCT
  GroupStatusValid,
  GroupStatusBusy,
  GroupMoving, 
  GroupHoming, 
  GroupErrorStop, 
  GroupNotReady, 
  GroupStandby, 
  GroupStopping,
 
  GroupDisabled, 
  AllAxesStanding, 
  ConstantVelocity, 
  Accelerating, 
  Decelerating, 
  InPosition, 
  GroupError					  : BIT; 

  GroupErrorId					: UDINT;

  AxisCount      				: UDINT;
  AxisCountEnabled      : UDINT;

  {attribute 'displaymode':='hex'}
  CaGroupOID            : OTCID;

  CaGroupState          : E_CA_GROUP_STATE;
END_STRUCT
END_TYPE

// ---- XTS_TRANSPORT/Mover/types/E_MOVER_CTRL.TcDUT
{attribute 'qualified_only'}
{attribute 'strict'}
{attribute 'to_string'}
TYPE E_MOVER_CTRL :
(
  MOVER_NULL,               // initial value at startup, used for change of order or retrigger
  MOVER_ENABLE,             // sets MC_Power.Enable
  MOVER_DISABLE,            // removes MC_Power.Enable
  MOVER_MOVE_TO_POS,        // modulo absolute positioning with MC_MoveAbsolute, InTargetPosition check
  MOVER_MOVE_TO_POS_CA,     // modulo absolute positioning with MC_MoveAbsoluteCA, InTargetPosition check
  MOVER_SEND_TO_POS_CA,     // modulo absolute positioning with MC_MoveAbsoluteCA, done after moving ReleaseDistance
  MOVER_HALT,               // halts mover; by use of MC_Halt mover is set passive in CA group
  MOVER_GEAR_IN,            // GearIn for mover in standstill

  MOVER_GEAR_IN_POS_CA,     // GearInPosCA of mover; when FB_GearInPosCa is InSync --> order is done; check SyncDistance yourself and release mover with e_mover_order.mover_SendToPos
  MOVER_GEAR_OUT,           // gear out for mover
  MOVER_RESET,              // MC_RESET for mover
  MOVER_INFO                // used to display MoverInfo in ST_MOVER_SELECTOR_STATE.Info
)UINT;
END_TYPE

// ---- XTS_TRANSPORT/Mover/types/E_MOVER_STATE.TcDUT
{attribute 'qualified_only'}
{attribute 'to_string'}
TYPE E_MOVER_STATE :
(
  MOVER_NULL,               // initial value at startup, used for change of order or retrigger
  MOVER_ENABLE,             // sets MC_Power.Enable
  MOVER_DISABLE,            // removes MC_Power.Enable
  MOVER_MOVE_TO_POS,        // modulo absolute positioning with MC_MoveAbsolute, InTargetPosition check
  MOVER_MOVE_TO_POS_CA,     // modulo absolute positioning with MC_MoveAbsoluteCA, InTargetPosition check
  MOVER_SEND_TO_POS_CA,     // modulo absolute positioning with MC_MoveAbsoluteCA, done after moving ReleaseDistance
  MOVER_HALT,               // halts mover; by use of MC_Halt mover is set passive in CA group
  MOVER_GEAR_IN,            // GearIn for mover in standstill

  MOVER_GEAR_IN_POS_CA,     // GearInPosCA of mover; when FB_GearInPosCa is InSync --> order is done; check SyncDistance yourself and release mover with e_mover_order.mover_SendToPos
  MOVER_GEAR_OUT,           // gear out for mover
  MOVER_RESET,              // MC_RESET for mover
  MOVER_INFO
)UINT;
END_TYPE

// ---- XTS_TRANSPORT/Mover/types/ST_GEAR_DATA.TcDUT
{attribute 'pack_mode' := '2'}
TYPE ST_GEAR_DATA :
STRUCT
  rDeltaToMasterPos       : LREAL;
  rModuloSyncPosSlave     : LREAL;
  rMasterStartDistance    : LREAL;
  rGearNumerator          : LREAL;
  iGearDenumerator        : USINT  := 1;
END_STRUCT
END_TYPE

// ---- XTS_TRANSPORT/Mover/types/ST_MOVER_CTRL.TcDUT
{attribute 'pack_mode' := '2'}
TYPE ST_MOVER_CTRL :
STRUCT
  Cmd             : E_MOVER_CTRL;  // order to execute on mover
END_STRUCT
END_TYPE

// ---- XTS_TRANSPORT/Mover/types/ST_MOVER_INFO.TcDUT
{attribute 'pack_mode' := '2'}
TYPE ST_MOVER_INFO :
STRUCT
  bMoverEnabled           : BIT;    // Axis[i].Status.ControlLoopClosed
  bMoverError             : BIT;    // Axis[i].Status.Error
  bMoverCoupled           : BIT;    // Axis[i].Status.Coupled OR _fbGearInPosCa[i].InSync
  bMoverStandstill        : BIT;    // Axis[i].Status.NotMoving
  bMoverAvoidingCollision : BIT;    // Axis[i].NcToPlc.StateDWord2.0
  bMoverInTarget          : BIT;    // Axis[i].NcToPlc.ActPos == rLastSetPos[i]

  rModuloActPos           : LREAL;  // Axis[i].NcToPlc.ModuloActPos
  rAbsActPos              : LREAL;  // Axis[i].NcToPlc.ActPos
  rAbsTargetPos           : LREAL;  // rLastSetPos[i]
  rModuloTargetPos        : LREAL;  // Tc2_Math.LMOD(_rLastSetPos[i], _RailLength)

  nErrorId                : UDINT;
END_STRUCT
END_TYPE

// ---- XTS_TRANSPORT/Mover/types/ST_MOVER_SELECTOR_STATE.TcDUT
TYPE ST_MOVER_SELECTOR_STATE :
STRUCT
  MoverIndex  : UINT;
  AxisId      : UDINT;
  State       : ST_MOVER_STATE;

  Info        : ST_MOVER_INFO;
END_STRUCT
END_TYPE

// ---- XTS_TRANSPORT/Mover/types/ST_MOVER_STATE.TcDUT
{attribute 'pack_mode' := '2'}
TYPE ST_MOVER_STATE :
STRUCT
  State           : E_MOVER_STATE;  // ST_MOVER_CTRL.Cmd with added E_PROGRESS
  MasterId        : USINT;            // mirror NC AxisId of Master axis
END_STRUCT
END_TYPE

// ---- XTS_TRANSPORT/Mover/types/ST_MOVE_DATA.TcDUT
{attribute 'pack_mode' := '2'}
TYPE ST_MOVE_DATA :
STRUCT
  // HAUD 2024 03 14
  // some init data added for example
  rPos            : LREAL :=   2275.0;
  rVelo           : LREAL :=    500.0;
  rAcc            : LREAL :=   5000.0;
  rJerk           : LREAL := 500000.0;
  rGap            : LREAL :=    100.0;
  rOverride       : LREAL :=    100.0;
  rDelta          : LREAL :=      0.05;
  rDistance       : LREAL :=     25.0;
END_STRUCT
END_TYPE

// ---- XTS_TRANSPORT/XtsStation/types/E_STATION_CHECK.TcDUT
{attribute 'qualified_only'}
{attribute 'strict'}
{attribute 'to_string'}
TYPE E_STATION_CHECK :
(
	CHECK_NULL,
  STATION_ID_INVALID := 9000,
  REFERENCE_CTRL_INVALID,
  REFERENCE_STATE_INVALID,
  REFERENCE_LIST_ITF_INVALID,
  REFERENCE_MOVER_ITF_INVALID,
  REFERENCE_MOVER_OFFSET_INVALID,
  REFERENCE_PARAMETER_INVALID,
  REFERENCE_MOVER_AXIS_REF_INVALID,

  REFERENCE_MASTER_AXIS_REF_INVALID,
  REFERENCE_GEAR_DATA_INVALID,
  REFERENCE_GEAR_PARAMETER_INVALID,

  CHECK_DONE    := 10_000
);
END_TYPE

// ---- XTS_TRANSPORT/XtsStation/types/E_STATION_CTRL.TcDUT
{attribute 'qualified_only'}
{attribute 'strict'}
{attribute 'to_string'}
TYPE E_STATION_CTRL :
(
  STATION_CTRL_NULL,              // nothing happens here
	STATION_INIT            := 1,   // hard reset of station, list is cleared
  STATION_DISABLE         := 10,  // 
  STATION_ENABLE,                 // 

  STATION_MOVER_ENTER     := 20,  // mover may enter station
  STATION_MOVER_ENTER_RETRY,      // retry after E_STATION_STATE.STATION_ERROR_INFEED_ERROR
  STATION_MOVER_SEND,             // do not enter, send to E_STATION_STATE.STATION_MOVER_OUT

  STATION_PROCESS_START   := 30,  // double handshake with extern
  STATION_PROCESS_DONE,           // single handshake with extern
  STATION_PROCESS_NEST_SKIP,

  STATION_MOVER_OUT       := 50,  // mover may leave station now; ticket for mover is checked here (ST_STATION_CTRL.nTargetStation)
  STATION_MOVER_OUT_RETRY,        // retry after E_STATION_STATE.STATION_ERROR_OUTFEED_ERROR

  STATION_MOVER_GONE      := 60   // mover has left station, last handshake station is empty

)USINT;
END_TYPE

// ---- XTS_TRANSPORT/XtsStation/types/E_STATION_GEAR_DISTANCE_AXIS.TcDUT
{attribute 'qualified_only'}
{attribute 'strict'}
{attribute 'to_string'}
TYPE E_STATION_GEAR_DISTANCE_AXIS :
(
  // which axis nSync distance is checked for termination of GearInPosCA.
  // after nSync distance the station does a regular outfeed to target station
	FOLLOW_THE_MASTER,
  FOLLOW_THE_SLAVE
)UINT;
END_TYPE

// ---- XTS_TRANSPORT/XtsStation/types/E_STATION_STATE.TcDUT
{attribute 'qualified_only'}
{attribute 'to_string'}
TYPE E_STATION_STATE :
(
	STATION_NO_INIT,                // startup state after power on, first cycle Init of station, switches to INIT when done

  STATION_INIT,                   // CONTINUE to DISABLE
                                  // State.MoverId deleted

  STATION_DISABLE         := 10,  // + CTRL.STATION_ENABLE  --> CONTINUE to DETECT_MOVER 
                                  // station is empty, no mover is handled, check enable from ctrl

  STATION_ENABLE,                 // init of work vars, check enable from ctrl

  STATION_DETECT_MOVER,           // (QueueCount > 0)       --> CONTINUE to MOVER_ENTER

  STATION_MOVER_ENTER     := 20,  // + CTRL.MOVER_ENTER     --> CONTINUE to PROCESS_START
                                  // + CTRL.MOVER_SEND      --> CONTINUE to MOVER_OUT
                                  // mover asking for entry

  STATION_MOVER_IN_TARGET,        // (MoveToPos==TRUE)      --> CONTINUE to PROCESS_START
                                  // mover is moving to PosWait + PosStop[_nNest]

  STATION_PROCESS_START   := 30,  // + CTRL.PROCESS_START   --> CONTINUE to PROCESS_START
                                  // + CTRL.PROCESS_DONE    --> CONTINUE to CHECK
                                  // wait until process started

  STATION_PROCESS_DONE,           // + CTRL.PROCESS_DONE    --> CONTINUE to CHECK
                                  // wait until process done

  STATION_CHECK           := 40,  // check for next nest in mask, 
                                  // (mask<>0) --> CHECK_NEST
                                  // (mask==0) --> MOVER_OUT

  STATION_CHECK_NEST,             // + CTRL.MOVER_ENTER     --> CONTINUE to MOVER_IN_TARGET
                                  // get next nest position

  STATION_MOVER_OUT       := 50,  // + CTRL.MOVER_OUT       --> CONTINUE to MOVER_RELEASE
                                  // mover asking to leave

  STATION_MOVER_RELEASE,          // (MoverSendToPos==TRUE) --> CONTINUE to MOVER_GONE
                                  // mover is released + check if release distance is passed

  STATION_MOVER_WRITE_TARGET,     // worker state to write mover ticket

  STATION_MOVER_GONE      := 60,  // + CTRL.MOVER_GONE      --> CONTINUE to INIT
                                  // mover out of station, enter mover in target station list


  STATION_ERROR_NULL      := 127,
  STATION_ERROR_LIST_GET_HEAD_FAULT,    // fatal error in linked list, must never occurr, must be debugged
  STATION_ERROR_LIST_REMOVE_HEAD_FAULT, // fatal error in linked list, must never occurr, must be debugged
  STATION_ERROR_LIST_ADD_TAIL_FAULT,    // fatal error in linked list, must never occurr, must be debugged

  STATION_ERROR_LIST_STATION_ID_WRONG,  // ticket data in Queue contains wrong Station Id, can be overruled by ctrl

  STATION_ERROR_LIST_MOVER_ID_INVALID,  // fatal error in ticket data, MoverId is out of range, must be fixed by ctrl, must be debugged

  STATION_ERROR_INFEED_ERROR,           // motion error during movement, retry must be triggered by ctrl
  STATION_ERROR_OUTFEED_ERROR,          // motion error during movement, retry by ctrl OR leave by ctrl

  STATION_ERROR_OUTFEED_TARGET_INVALID, // ticket data for nTargetStation is not plausible, can be fixed by ctrl

  STATION_ERROR_FATAL     := 255 // the thing that must not be, all fatal errors end up here
)USINT;
END_TYPE

// ---- XTS_TRANSPORT/XtsStation/types/E_STATION_TYPE.TcDUT
{attribute 'qualified_only'}
{attribute 'strict'}
{attribute 'to_string'}
TYPE E_STATION_TYPE :
(
	INVALID,
  STATION_PROCESS,      // default station with/without process
  STATION_GEAR_IN_POS   // GearInPos station for flying saw with MasterAxis
)USINT;
END_TYPE

// ---- XTS_TRANSPORT/XtsStation/types/ST_STATION_CTRL.TcDUT
{attribute 'pack_mode' := '2'}
TYPE ST_STATION_CTRL :
STRUCT
  Cmd             : E_STATION_CTRL;
  {attribute 'displaymode':='bin'}
  nMask           : BYTE;           // nest mask for sending mover to next station
  nTargetStation  : USINT;          // where to next?
  rOffset         : REAL;           // optional offset for mover in target station when leaving sending station; 
                                    // use case: position correction of workpiece on wpc by vision
END_STRUCT
END_TYPE

// ---- XTS_TRANSPORT/XtsStation/types/ST_STATION_GEAR_PARAMETER.TcDUT
TYPE ST_STATION_GEAR_PARAMETER :
STRUCT
  eDistance           : E_STATION_GEAR_DISTANCE_AXIS; // follow which leader?
  rSyncDistance       : LREAL := 100.0;               // synchrone distance while the mover is geared in
  rMinDistanceToSync  : LREAL := 100.0;               // minimum distance for mover to get nSync with the Master
END_STRUCT
END_TYPE

// ---- XTS_TRANSPORT/XtsStation/types/ST_STATION_LIST_RESULT.TcDUT
TYPE ST_STATION_LIST_RESULT :
STRUCT
  wState    : WORD;   // wState == 0 --> all ok
  nIndex    : ULINT;
  stData    : ST_STATION_MOVER_DATA;  // copy of list entry
END_STRUCT
END_TYPE

// ---- XTS_TRANSPORT/XtsStation/types/ST_STATION_MOVER_DATA.TcDUT
{attribute 'pack_mode' := '2'}
TYPE ST_STATION_MOVER_DATA :
STRUCT
  nMoverId        : USINT;  // who am I?  !! MUST be correct !! - movement to base position sets everything in order, DO NOT manipulate!
  nTargetStation  : USINT;  // where shall I be? used for double checking with StationId at infeed of mover into station

  {attribute 'displaymode':='bin'}
  nMask           : BYTE;   // how many of you are there? (1 = default, no action required)

  rOffset         : REAL;   // offset for use in work flow !! added to static mover offset for every nest(bit) in nMask!!
END_STRUCT
END_TYPE

// ---- XTS_TRANSPORT/XtsStation/types/ST_STATION_PARAMETER.TcDUT
TYPE ST_STATION_PARAMETER :
STRUCT
  eType             : E_STATION_TYPE := 1;  // StationProcess or StationGearInPos
  sText             : STRING(80);           // only description
  rPosWait          : REAL;                 // start of station, 
                                            // a sending station is using this value 
                                            // to send mover to

  rReleaseDistance  : REAL;                 // distance mover has to travel (from ActPos) 
                                            // in order for station to go back to disable

  rGap              : REAL;
  rVelo             : REAL;
  rAccDec           : REAL;
  rJerk             : REAL;

  // how many nests (stop positions) mover has to stop at (1 = default)
  nConfiguredStopCount  : USINT := 1; // 1-8 --> NestMask = BYTE

  // mover stop position in station, relative to rPosWait!!
  rPosStop          : ARRAY[1..8] OF LREAL;
END_STRUCT
END_TYPE

// ---- XTS_TRANSPORT/XtsStation/types/ST_STATION_STATE.TcDUT
{attribute 'pack_mode' := '2'}
TYPE ST_STATION_STATE :
STRUCT
  State           : E_STATION_STATE;
  {attribute 'displaymode':='bin'}
  nMask           : BYTE;
  nMoverId        : USINT;
  rMoverModPos    : LREAL;            // modulo position of detected mover
  nQueue          : USINT;            // queue count for station
END_STRUCT
END_TYPE

// ---- XTS_TRANSPORT/XtsStation/types/T_NEST_OFFSET.TcDUT
TYPE T_NEST_OFFSET : ARRAY[1..MAX_MOVER]        OF
                     ARRAY[1..MAX_STATION_NEST] OF LREAL;
END_TYPE

// ---- XTS_TRANSPORT/_Visualization/types/ST_XPU_STRINGS.TcDUT
TYPE ST_XPU_STRINGS :
STRUCT
  sXpuState       ,
  sXpuResult      ,
  sXpuCyclicCheck ,
  sXpuOpMode      ,
  sXpuMoverId_DetectionMode,
  sXpuMoverPosAssignement : STRING(30) := 'NULL';
END_STRUCT
END_TYPE

// ---- XTS_TRANSPORT/Xpu/types/E_XPU_CHECK.TcDUT
{attribute 'qualified_only'}
{attribute 'to_string'}
TYPE E_XPU_CHECK :
(
  INIT_CHECK,
  INIT_CHECK_ERROR,
  START_CHECK,
  XPU_INSTANCE_NULL,
  XPU_RAIL_LENGTH,
  GROUP_RAIL_LENGTH,
  RAIL_LENGTH_COMPARE,
  GROUP_NOT_CONFIGURED,
  GROUP_OID_MISMATCH,

  MOVER_COUNT             := 10,
  MOVER_COUNT_ZERO,
  MOVER_COUNT_NOT_EQUAL,

  PROCESSING_UNIT_POSITIONS_VALID         := 20,
  PROCESSING_UNIT_GET_DATA_EXCEED,

  MOVER_ID_STANDARD       := 30,
  MOVER_ID_SIMULATION,
  MOVER_ID_DETECTION_MODE,
  MOVER_ID_DETECTION_VALID,
  MOVER_ID_DETECTION_DC_LINK,
  MOVER_ID_DETECTION_BUSY,
  MOVER_ID_DETECTION_IDLE,
  MOVER_ID_DETECTION_STATE,
  MOVER_ID_MULTIPLE_NOT_SUPPORTED,

  POINTER_CHECK           := 90,
  POINTER_NULL_CTRL,
  POINTER_NULL_STATE,

  CHECK_DONE      := 10_000
)UINT;
END_TYPE

// ---- XTS_TRANSPORT/Xpu/types/E_XPU_CTRL.TcDUT
{attribute 'strict'}
TYPE E_XPU_CTRL :
(
  XTS_CMD_NULL,
  XTS_CMD_INIT                  := 10,
  //XTS_CMD_READ_STN_CONFIG       := 20,
  XTS_IDLE                      := 30
)UINT;
END_TYPE

// ---- XTS_TRANSPORT/Xpu/types/E_XPU_INIT.TcDUT
{attribute 'to_string'}
TYPE E_XPU_INIT :
(
	INIT_START,
  INIT_ENVIRONMENT_OID            := 10,
  INIT_INFO_SERVER_ITF,
  INIT_INFO_SERVER_STATION_COUNT,
  INIT_INFO_SERVER_STATION_OID,
  INIT_CA_GROUP_OID               := 20,
  INIT_CA_GROUP_GET_OID,
  INIT_CA_GROUP_CHECK_OID,
  INIT_CA_GROUP_COM,
  INIT_PARAMETERSET_COUNT,
  INIT_PARAMETERSET_OID,
  INIT_PARAMETERSET_COM,
  INIT_PARAMETERSET_COM_INIT,
  INIT_PARAMETERSET_COM_NEXT,
  INIT_PROCESSING_UNIT_COM        := 30,
  INIT_PROCESSING_UNIT_COM_INIT,
  INIT_PROCESSING_UNIT_PART_COUNT,
  INIT_PROCESSING_UNIT_PART_OID,
  INIT_PROCESSING_UNIT_TRACK_COUNT,
  INIT_PROCESSING_UNIT_TRACK_OID,
  INIT_PROCESSING_UNIT_MOVER_COUNT,
  INIT_PROCESSING_UNIT_MOVER_OID,
  INIT_PROCESSING_UNIT_TASK_COUNT,
  INIT_PROCESSING_UNIT_TASK_OID,
  INIT_TRACK_COM                  := 50,
  INIT_TRACK_COM_INIT,
  INIT_PART_COM                   := 60,
  INIT_PART_COM_INIT,
  INIT_PART_MODULE_COUNT,
  INIT_PART_MODULE_OID,
  INIT_PART_MODULE_COM,
  INIT_PART_MODULE_COM_INIT,
  INIT_PART_MODULE_COM_NEXT,
  INIT_MOVER_COM                  := 70,
  INIT_MOVER_COM_INIT,
  INIT_MOVER_COM_NEXT,
  INIT_NCT_CONTROLLER_OID         := 80,
  INIT_NCT_CONTROLLER_COM,
  INIT_NCT_CONTROLLER_COM_INIT,
  INIT_NCT_BASE_UNIT_COUNT,
  INIT_NCT_BASE_UNIT_ITF,
  INIT_NCT_BASE_UNIT_NEXT,
  INIT_DATA_GET                   := 90,
  INIT_DATA_CHECK,
  INIT_DONE                       := 100
)UINT;
END_TYPE

// ---- XTS_TRANSPORT/Xpu/types/E_XPU_STATE.TcDUT
{attribute 'to_string'}
TYPE E_XPU_STATE :
(
  XTS_NULL,
  XTS_INVALID,
  XTS_INIT                      := 10,    // initialize XPU
  XTS_STATION_INFO_READ         := 20,    // get Station information from Xpu
  XTS_IDLE                      := 30
)UINT;
END_TYPE

// ---- XTS_TRANSPORT/Xpu/types/ST_XPU_CTRL.TcDUT
{attribute 'pack_mode' := '2'}
TYPE ST_XPU_CTRL :
STRUCT
  Cmd             : E_XPU_CTRL;
END_STRUCT
END_TYPE

// ---- XTS_TRANSPORT/Xpu/types/ST_XPU_INFO.TcDUT
{attribute 'pack_mode' := '2'}
TYPE ST_XPU_INFO :
STRUCT
  AllPositionsValid   : BIT;
  IdDetectionError    : BIT;
  IdDetectionValid    : BIT;
  IdDetectionActive   : BIT;

  OperationMode       : UINT;

  IdDetectionMode           : UINT;
  MoverPositionAssignement  : UINT;

  nDetectedAxisCount  : UINT;
  nExpectedAxisCount  : UINT;

  nParameterSetCount  : UINT;
  nModuleCount        : UINT;
  rRailLength         : LREAL;
END_STRUCT
END_TYPE

// ---- XTS_TRANSPORT/Xpu/types/ST_XPU_STATE.TcDUT
{attribute 'pack_mode' := '2'}
TYPE ST_XPU_STATE :
STRUCT
  Init            : E_XPU_INIT;
  State           : E_XPU_STATE;
  Check           : E_XPU_CHECK;  // cyclic check result
  DcLink          : BIT;          // power all motor modules is ON
END_STRUCT
END_TYPE

// ---- XTS_TRANSPORT/XtsTransportUnit/types/E_XTS_TRANSPORT_CHECK.TcDUT
{attribute 'qualified_only'}
{attribute 'to_string'}
TYPE E_XTS_TRANSPORT_CHECK :
(
  // info for cyclic checks
  INIT_CHECK,
  START_CHECK,    // check cycle start
  XPU_INIT,       // Xpu: initialization


  // errors in fb_TransportUnit.Check()
  POINTER_CHECK           := 9000,
  POINTER_NULL_CTRL,

  POINTER_NULL_STATE,
  POINTER_NULL_XPU_CTRL,

  POINTER_NULL_XPU_STATE,
  POINTER_NULL_XPU_INFO,

  POINTER_NULL_GROUP_ITF,
  POINTER_NULL_GROUP_INFO,

  POINTER_NULL_MOVER,
  POINTER_NULL_MOVER_ITF,

  POINTER_NULL_MOVER_INFO,
  POINTER_NULL_MOVER_LAST_POS,
  POINTER_NULL_MOVER_LAST_GAP,

  POINTER_NULL_STATION_START,
  POINTER_NULL_STATION_ITF,
  POINTER_NULL_STATION_CONTROL,
  POINTER_NULL_STATION_STATE,
  POINTER_NULL_STATION_CTRL_ITF,

  DONE_CHECK              := 10000
)UINT;
END_TYPE

// ---- XTS_TRANSPORT/XtsTransportUnit/types/E_XTS_TRANSPORT_CTRL.TcDUT
{attribute 'strict'}
{attribute 'to_string'}
TYPE E_XTS_TRANSPORT_CTRL :
(
  CMD_NULL,
  CMD_INIT                  := 10,  // Xpu, Group, Mover initialization: clear errors, clear group, check Xpu data, check mover detection
  CMD_IDLE,

  CMD_MOVER_ENABLE          := 20,  // all mover are enabled, checked for ControlLoopClosed
  CMD_MOVER_DISABLE,                // all mover are disabled, no axis in CaGroup: no error, any axis in CaGroup: group error
  CMD_MOVER_HALT_CA,                // all movers are stopped with MC_HaltCA[]. ONLY use if all movers are in CA group
  CMD_MOVER_STOP,

  CMD_GROUP_CLEAR           := 30,  // halt all movers, clear errors, remove all movers from group, clear group
  CMD_GROUP_BUILD,                  // add all movers to group
  CMD_GROUP_ENABLE,                 // group with movers is enabled
  CMD_GROUP_STOP,                   // moving CA Group is stopped

  CMD_TRANSPORT_START       := 40,  // move all mover[i] to start position
  CMD_TRANSPORT_RESTART             // move all mover[i] to LastPosition[i]

)UINT;
END_TYPE

// ---- XTS_TRANSPORT/XtsTransportUnit/types/E_XTS_TRANSPORT_STATE.TcDUT
{attribute 'to_string'}
TYPE E_XTS_TRANSPORT_STATE :
(
  TRANSPORT_NULL,
  TRANSPORT_INVALID,
  TRANSPORT_INIT            := 10,  // Xpu, Group, Mover initialization: init TcCOM objects, clear errors, clear group, check Xpu data, check mover detection
  TRANSPORT_IDLE,                   // cyclic check for errors, check Xpu data

  TRANSPORT_MOVER_ENABLE    := 20,  // all mover are enabled, checked for ControlLoopClosed
  TRANSPORT_MOVER_DISABLE,          // all mover are disabled
  TRANSPORT_MOVER_HALT_CA,          // all mover standstill
  TRANSPORT_MOVER_STOP,

  TRANSPORT_GROUP_CLEAR     := 30,  // halt all movers, clear errors, remove all movers from group, clear group
  TRANSPORT_GROUP_BUILD,            // add all movers to group
  TRANSPORT_GROUP_ENABLE,           // group with movers is enabled
  TRANSPORT_GROUP_STOP,             // CaGroup Stop, CaGroup Reset, All movers halt

  TRANSPORT_START           := 40,  // move all mover[i] to start position
  TRANSPORT_RESTART                 // move all mover[i] to LastPosition[i]
)UINT;
END_TYPE

// ---- XTS_TRANSPORT/XtsTransportUnit/types/ST_XTS_TRANSPORT_CTRL.TcDUT
{attribute 'pack_mode' := '2'}
TYPE ST_XTS_TRANSPORT_CTRL :
STRUCT
  Cmd       : E_XTS_TRANSPORT_CTRL;
END_STRUCT
END_TYPE

// ---- XTS_TRANSPORT/XtsTransportUnit/types/ST_XTS_TRANSPORT_STATE.TcDUT
{attribute 'pack_mode' := '2'}
TYPE ST_XTS_TRANSPORT_STATE :
STRUCT
  State         : E_XTS_TRANSPORT_STATE;  // combined value of state and result(e_progress); (hint: extract state value by mod division)
  Check         : E_XTS_TRANSPORT_CHECK;

  XpuState      : ST_XPU_STATE;
  XpuInfo       : ST_XPU_INFO;
  GroupInfo     : ST_GROUP_INFO; 
END_STRUCT
END_TYPE

// ---- APPLICATION/GVL_APPLICATION.TcGVL
VAR_GLOBAL CONSTANT
  // These my be the number of processes YOU require
  MAX_PROCESS       : E_INSTANCE := E_INSTANCE.INSTANCE_MAX;
END_VAR
{attribute 'qualified_only'}
VAR_GLOBAL
  //-----------------------------------------------------------------------------------------------
  // APPLICATION territory, your territory
  //
  //  - here you find diplomats for building transport logic:
  //
  //    - for grouping of stations
  //      - multiplication of single stations into processes vis ProcessCollector
  //      - dedicated transport procedures by extending fb_Instance
  //        - transport procedure on this level always uses a ProcessCollector
  //
  //    - for a cyclic process ticket list
  //      - input for process tickets via any network or protocol
  //
  //    - for a process ticket conductor
  //      - distributes process tickets to process index
  //-----------------------------------------------------------------------------------------------
  //-----------------------------------------------------------------------------------------------
  // Linked List instances
  //-----------------------------------------------------------------------------------------------
  ProcessList           : ARRAY[1..MAX_PROCESS] OF fb_Process_LinkedList; // information transfer between processes
  ItfProcessList        : ARRAY[1..MAX_PROCESS] OF I_Process_LinkedList;  // use this interface in your function blocks
  //-----------------------------------------------------------------------------------------------
  //-----------------------------------------------------------------------------------------------
  // Collector instances
  //
  //  - layer for grouping parallel XtsStations for process handshakes
  //-----------------------------------------------------------------------------------------------
  //  - fb_ProcessCollector:
  //    - uses .ProcessCtrl and .ProcessState for handshakes with application
  //
  //    - .ActivateStation is evaluated after enabling infeed in state 
  //      E_PROCESS_STATE.PROCESS_DISABLE:/E_PROGRESS.PROGRESS_BUSY:
  //      
  //    - ST_PROCESS_STATE:
  //      - contains 3 enumerations for you to check
  //      - State           : E_PROCESS_STATE;
  //        - main state for handshakes
  //
  //      - Result          : E_PROGRESS;
  //        - substate for checks during handshake; 
  //          PROGRESS_BUSY --> handshakes are accepted (see fb_ProcessCollecotr.Cycle())
  //
  //      - Check           : E_PROCESS_CHECK;
  //        - cyclic pointer check: use this on startup of your application
  //
  //    - inherits fb_StationCollector
  //-----------------------------------------------------------------------------------------------
  //-----------------------------------------------------------------------------------------------
  ProcessCollector      : ARRAY[1..MAX_PROCESS] OF fb_ProcessCollector;       // grouping of XtsStations
  ItfProcessCollector   : ARRAY[1..MAX_PROCESS] OF I_ProcessCollector;        // interface for use in your function blocks like BufferInfeed etc.
  //-----------------------------------------------------------------------------------------------
  // cyclic linked lists
  //
  //  - fb_LinkedListCtrl
  //    - is controlled via Ctrl/State pair
  //    - provides I_Process_LinkedList for use in conected class
  //-----------------------------------------------------------------------------------------------
  TicketList            : fb_Process_LinkedListCtrl;
  TicketListControl     : ST_LIST_CTRL;
  TicketListState       : ST_LIST_STATE;
  TicketListDataInput   : ST_LIST_NODE_DATA;   // datafield for you to write(add) your data
  TicketListDataOutput  : ST_LIST_NODE_DATA;   // datafield for you to read (get) your data
  //-----------------------------------------------------------------------------------------------
  //-----------------------------------------------------------------------------------------------
  // Distribution of LinkedList ticket
  //
  //  - fb_ProcessConductor extends fb_Instance
  //    - is controlled via instance Ctrl/State pair
  //    - consumes I_Process_LinkedList for moving 
  //      the ticket from the cyclic list into the process list of ST_PROCESS_DATA.nProcessId
  //-----------------------------------------------------------------------------------------------
  ProcessConductor      : fb_ProcessConductor;
  //-----------------------------------------------------------------------------------------------
  //-----------------------------------------------------------------------------------------------
  // Configuration of XtsTransport
  //
  //  - fb_Configuration stores data in xml format
  //    - is controlled via data Ctrl/State pair
  //-----------------------------------------------------------------------------------------------
  StationConfig         : fb_Configuration;
  ConfigCtrl            : ST_DATA_CTRL;
  ConfigState           : ST_DATA_STATE;
  //-----------------------------------------------------------------------------------------------
  //-----------------------------------------------------------------------------------------------
  // static mover offsets XtsTransport
  //
  //  - fb_MoverPositionOffsetData stores data in xml format
  //    - is controlled via data Ctrl/State pair
  //-----------------------------------------------------------------------------------------------
  MoverOffsetsData      : fb_MoverPositionOffsetData;
  OffsetDataCtrl        : ST_DATA_CTRL;
  OffsetDataState       : ST_DATA_STATE;
  //-----------------------------------------------------------------------------------------------
END_VAR

// ---- _MSG/GVL_MSG_AXIS.TcGVL
{attribute 'qualified_only'}
VAR_GLOBAL CONSTANT
  //-----------------------------------------------------------------------------
  // file paths for message system
  //  - compiler define option WIN switches to Windows file paths
  //-----------------------------------------------------------------------------
{IF defined (WIN)}
  {info 'PLC_MOTION_LAYER: WIN'}
  LOG_DIR               : STRING  := 'C:\TwinCAT\#MsgFiles\';
{ELSE}
  {info 'PLC_MOTION_LAYER: BSD'}
  LOG_DIR               : STRING  := '/usr/local/etc/TwinCAT/#MsgFiles/';
{END_IF}

  LOG_FILE              : STRING  := concat(TO_STRING(TwinCAT_SystemInfoVarList._AppInfo.AdsPort), '_MSG_PLC_');
  LOG_FILE_METRIC       : STRING  := concat(TO_STRING(TwinCAT_SystemInfoVarList._AppInfo.AdsPort), '_MSG_Metrics_');
END_VAR
VAR_GLOBAL
  //-----------------------------------------------------------------------------
  // Message System
  //  - Everybody uses f_MessageSet(ST_Message)
  //    - DECISION WHICH LIST IS MADE IN f_MessageSet !!
  //    - which list to use is determined by e_Device in your message
  //
  //  - MessageData instances are self sufficient and need only 
  //    datafield assignment for correct data-flow
  //
  //
  //-----------------------------------------------------------------------------
  //-----------------------------------------------------------------------------
  //-----------------------------------------------------------------------------
  // (ST_Message.eDevice := from Device_Null to XfcAxis)
  //-----------------------------------------------------------------------------
  MotionMessageData               : fb_MessageDataCtrl;
  MotionMessageCtrl               : st_message_ctrl;
  MotionMessageState              : st_message_state;

  MotionMessages                  : ARRAY[1..GVL_MSG_XTS.MAX_MESSAGE] OF ST_Message;
  MessageMotionIndex              : UINT := 0; // message index for base layer
  MessageMotionError              : UINT := 0; // error counter for base layer
  //-----------------------------------------------------------------------------
  //-----------------------------------------------------------------------------
  // (ST_Message.eDevice := e_Device.Metrics)
  //-----------------------------------------------------------------------------
  MetricMessageData               : fb_MessageDataCtrl;
  MetricMessageCtrl               : st_message_ctrl;
  MetricMessageState              : st_message_state;

  MetricMessages                  : ARRAY[1..GVL_MSG_XTS.MAX_MESSAGE] OF ST_Message;
  MessageMetricIndex              : UINT := 0; // message index for metrics data
  MessageMetricError              : UINT := 0; // error counter for metrics data
  //-----------------------------------------------------------------------------
  //-----------------------------------------------------------------------------
  fbLocalTime                     : fb_LocalTime;
  dtLocalTime                     : DT;
  sLocalTime                      : STRING;
  //-----------------------------------------------------------------------------
  //-----------------------------------------------------------------------------
  //-----------------------------------------------------------------------------
  //-----------------------------------------------------------------------------
{IF defined (TEST)}
  {info 'TEST logging enabled'}
  MessageLevel                    : E_MessageType := eMessageverbose; // a lot of messages
{ELSE}
  MessageLevel                    : E_MessageType := eMessageEmpty; // only errors are written into list 
{END_IF}

  MessageLevelAxisPtp             : ARRAY[1..PLC_CONSTANT.MAX_AXIS]   OF E_MessageType;
  MessageLevelAxisCam             : ARRAY[1..PLC_CONSTANT.MAX_AXIS]   OF E_MessageType;
  MessageLevelAxisFly             : ARRAY[1..PLC_CONSTANT.MAX_AXIS]   OF E_MessageType;
  MessageLevelNciChn              : ARRAY[1..PLC_CONSTANT.MAX_NCI_CH] OF E_MessageType;

  MessageLevelTriggerBox          : ARRAY[1..PLC_CONSTANT.MAX_TRIGGER_BOX]  OF E_MessageType;
  MessageLevelTouchProbe          : ARRAY[1..PLC_CONSTANT.MAX_TOUCH_PROBE]  OF E_MessageType;


  // diag data
  dbg_AxisIdxGearIn               : ARRAY[1..PLC_CONSTANT.MAX_AXIS]      OF BYTE; // diag for Axis gear in
  dbg_AxisIdxGearInMultiMaster    : ARRAY[1..PLC_CONSTANT.MAX_AXIS,1..4] OF BYTE; // diag for Axis gear in multi master
  dbg_AxisIdxCamIn                : ARRAY[1..PLC_CONSTANT.MAX_AXIS]      OF BYTE; // diag for Axis cam in
END_VAR

// ---- _MSG/GVL_MSG_XTS.TcGVL
{attribute 'qualified_only'}
VAR_GLOBAL CONSTANT
  //-----------------------------------------------------------------------------
  // file paths for message system
  //  - compiler define option WIN switches to Windows file paths
  //-----------------------------------------------------------------------------
{IF defined (WIN)}
  {info 'WIN folders'}
  LOG_DIR               : STRING  := 'C:\TwinCAT\#MsgFiles\';       // delimiter at the end is mandatory!!
  CON_DIR               : STRING  := 'C:\TwinCAT\#Configuration\';  // delimiter at the end is mandatory!!
{ELSE}
  {info 'BSD folders'}
  LOG_DIR               : STRING  := '/usr/local/etc/TwinCAT/#MsgFiles/';       // delimiter at the end is mandatory!!
  CON_DIR               : STRING  := '/usr/local/etc/TwinCAT/#Configuration/';  // delimiter at the end is mandatory!!
{END_IF}

  LOG_FILE              : STRING  := 'MSG_XtsTransport_';
  LOG_FILE_APP          : STRING  := 'MSG_Application_';
  LOG_FILE_METRIC       : STRING  := 'MSG_XtsTransportMetrics_';

  MAX_MESSAGE           : UINT    := 2000; // max entry in message list
END_VAR
VAR_GLOBAL
  //-----------------------------------------------------------------------------
  // Message System
  //  - Everybody uses f_MessageSet(ST_Message)
  //    - DECISION WHICH LIST IS MADE IN f_MessageSet !!
  //    - which list to use is determined by e_Device in your message
  //
  //  - MessageData instances are self sufficient and need only 
  //    datafield assignment for correct data-flow
  //
  //
  //-----------------------------------------------------------------------------
  //-----------------------------------------------------------------------------
  //-----------------------------------------------------------------------------
  // (ST_Message.eDevice := e_Device.Application)
  //----------------------------------------------------------------------------- 
  ApplicationMessageData          : fb_MessageDataCtrl;
  ApplicationMessageCtrl          : st_message_ctrl;
  ApplicationMessageState         : st_message_state;

  ApplicationMessages             : ARRAY[1..MAX_MESSAGE] OF ST_Message;
  MessageApplicationIndex         : UINT := 0; // message index for higher layers (grouping, Instances, etc.)
  MessageApplicationError         : UINT := 0; // error counter for higher learning
  //-----------------------------------------------------------------------------
  //-----------------------------------------------------------------------------
  // (ST_Message.eDevice := from Device_Null to XfcAxis)
  //-----------------------------------------------------------------------------
  TransportMessageData            : fb_MessageDataCtrl;
  TransportMessageCtrl            : st_message_ctrl;
  TransportMessageState           : st_message_state;

  TransportMessages               : ARRAY[1..MAX_MESSAGE] OF ST_Message;
  MessageTransportIndex           : UINT := 0; // message index for base layer
  MessageTransportError           : UINT := 0; // error counter for base layer
  //-----------------------------------------------------------------------------
  //-----------------------------------------------------------------------------
  // (ST_Message.eDevice := e_Device.Metrics)
  //-----------------------------------------------------------------------------
  MetricsMessageData              : fb_MessageDataCtrl;
  MetricsMessageCtrl              : st_message_ctrl;
  MetricsMessageState             : st_message_state;

  MetricsMessages                 : ARRAY[1..MAX_MESSAGE] OF ST_Message;
  MessageMetricsIndex             : UINT := 0; // message index for metrics data
  MessageMetricsError             : UINT := 0; // error counter for metrics data
  //-----------------------------------------------------------------------------
  //-----------------------------------------------------------------------------
  // (ST_Message.eDevice := e_Device.ProductData)
  //-----------------------------------------------------------------------------
  ProductMessageData              : fb_MessageDataCtrl;   // This is for you
  ProductMessageCtrl              : st_message_ctrl;
  ProductMessageState             : st_message_state;

  ProductMessages                 : ARRAY[1..MAX_MESSAGE] OF ST_Message;
  MessageProductIndex             : UINT := 0; // message index for your product data
  MessageProductError             : UINT := 0; // error counter for your product data
  //-----------------------------------------------------------------------------
  //-----------------------------------------------------------------------------
  fbLocalTime                     : fb_LocalTime;
  dtLocalTime                     : DT;
  sLocalTime                      : STRING;
  //-----------------------------------------------------------------------------
  //-----------------------------------------------------------------------------
  //-----------------------------------------------------------------------------
  //-----------------------------------------------------------------------------
  MessageLevelXpu                 : E_MessageType;
  MessageLevelStations            : ARRAY[1..MAX_STATION] OF E_MessageType;
  MessageLevelMovers              : ARRAY[1..MAX_MOVER]   OF E_MessageType;

  MessageLevelProcess             : ARRAY[1..MAX_PROCESS] OF E_MessageType;

{IF defined (TEST)}
  {info 'TEST logging enabled'}
  MessageLevel                    : E_MessageType := eMessageinfo; // a lot of messages
{ELSE}
  MessageLevel                    : E_MessageType := eMessageEmpty; // only errors are written into list 
{END_IF}

END_VAR

// ---- PLC_MOTION/_GVL/PLC_CONSTANT.TcGVL
//{attribute 'qualified_only'}
VAR_GLOBAL CONSTANT


  //-----------------------------------------------------------------------------
  // AXIS related limits
  //-----------------------------------------------------------------------------
  MAX_AXIS              : UINT    := 3;
  MAX_RETRY             : UINT    := 5;


  //-----------------------------------------------------------------------------
  // NCI related limits and *.nc standard folder
  //-----------------------------------------------------------------------------
{IF NOT defined (BSD)}
  NCI_DIR               : STRING  := 'C:\TwinCAT\Mc\Nci\';
{ELSE}
  NCI_DIR               : STRING  := '/usr/local/etc/TwinCAT/Mc/Nci/';
{END_IF}

{IF defined (NCI)}
  {info 'PLC_MOTION_LAYER: NCI'}
  NCI_ACTIVE            : BOOL    := TRUE;
  CONFIG_NAME           : STRING  := 'NCI_Spec_Ch_';
{ELSE}
  NCI_ACTIVE            : BOOL    := FALSE;
  CONFIG_NAME           : STRING  := 'NCI_NOT_ACTIVE';
{END_IF}

  MAX_NCI_CH            : UINT    := 1;

  MAX_PATH_STEPS        : UINT    := 5;
  MAX_MC_AXIS           : UINT    := 3;
  MAX_AUX_AXIS          : UINT    := 2;
  MAX_R_PARA            : UINT    := 10;


  //-----------------------------------------------------------------------------
  // CAMMING related limits
  //-----------------------------------------------------------------------------
{IF defined (CAM)}
  {info 'PLC_MOTION_LAYER: CAM'}
  CAM_ACTIVE                  : BOOL    := TRUE;
{ELSE}
  CAM_ACTIVE                  : BOOL    := FALSE;
{END_IF}

  MAX_CAM_CH                  : UINT    := 1;

  MAX_MOTION_FUNCTION_POINTS  : UINT    := 10;

  // HAUD
  // 17.07.2024
  // Start Implementation of Position Trigger function
  //  - Timestamp/position output
  //  - Latch DC time from input
  
  MAX_TRIGGER_BOX             : UINT := 12;
  MAX_TOUCH_PROBE             : UINT := 12;
  MAX_TRIGGER_COUNT           : UINT :=  4;
  MAX_MTI_CH                  : UINT :=  1; // MAX mti channel per EL terminal

{IF defined (XFC)}
  {info 'PLC_MOTION_LAYER: XFC'}
  XFC_ACTIVE                  : BOOL := TRUE;
{ELSE}
  XFC_ACTIVE                  : BOOL := FALSE;
{END_IF}

  // HAUD
  // 2026 05 28
  // Gear In Pos implementation for flying saw application 

{IF defined (SAW)}
  {info 'PLC_MOTION_LAYER: FLYING_SAW'}
  FLY_SAW_ACTIVE              : BOOL  := TRUE;
{ELSE}
  FLY_SAW_ACTIVE              : BOOL  := FALSE;
{END_IF}
END_VAR

// ---- XTS_TRANSPORT/GVL_XTS.TcGVL
{attribute 'qualified_only'}
VAR_GLOBAL
  //---------------------------------------------------------------------------
  // XTS Station
  //  - handshakes mover in station with extern control
  //  - station parameters (positions, gap, dyn. constraints, description...)
  StationStart        : ST_STATION_PARAMETER;   // Xts transport is sending all mover to this position (CMD_TRANSPORT_START)
  StationStartIndex   : UINT := 1;              // index of XtsStation where all movers are entered into linked list.

  // station handshaking with mover and extern process
  // station sends mover to target station/WaitPos
  // station adds mover data to LinkedList.AddTail() of target station
  Station             : ARRAY[1..MAX_STATION] OF fb_StationProcess;
  StationGearIn       : ARRAY[1..MAX_STATION] OF fb_StationGearInPos;

  StationList         : ARRAY[1..MAX_STATION] OF fb_Station_LinkedList;

  StationQueue        : ARRAY[1..MAX_STATION]    OF 
                        ARRAY[1..MAX_LIST_NODES] OF ST_STATION_MOVER_DATA;

  // interface for access to List methods
  StationListItf      : ARRAY[1..MAX_STATION] OF I_Station_LinkedList;

  // interface for access to station methods
  StationCtrlItf      : ARRAY[1..MAX_STATION] OF I_XtsTransport_Station;

  // ctrl / state datafields for extern control
  StationCtrl         : ARRAY[1..MAX_STATION] OF ST_STATION_CTRL;   // control for extern to write, you can do whatever you want as long as you do as I say
  StationState        : ARRAY[1..MAX_STATION] OF ST_STATION_STATE;  // state for extern to read, this is what I tell you to do

  // station parameter
  StationParameter    : ARRAY[1..MAX_STATION] OF ST_STATION_PARAMETER; // wherever, whenever you want. Build it and they will come...

  // station GearInPosCA parameter and data structs
  StationGearParameter: ARRAY[1..MAX_STATION] OF ST_STATION_GEAR_PARAMETER;
  StationGearData     : ARRAY[1..MAX_STATION] OF ST_GEAR_DATA;

  // static position offsets in stations
  PositionOffset      : ARRAY[1..MAX_STATION] OF T_NEST_OFFSET; // added to PosStop[] in XtsStation


  //---------------------------------------------------------------------------
  // XTS
  // XTS TransportUnit
  //  - This is ground control
  //  - handles request for XPU, Group, Mover, StartUp, ReStart
  XtsTransport        : fb_TransportUnit;         // manages members of XTS transport for extern to access

  XtsTransportCtrl    : ST_XTS_TRANSPORT_CTRL;    // control of XTS transport for extern to write
  XtsTransportState   : ST_XTS_TRANSPORT_STATE;   // state   of XTS transport for extern to read


  //---------------------------------------------------------------------------
  // XPU
  // XTS-Utility checks
  // XTS-Utility interfaces for you to use
  Xpu             : fb_XpuCtrl;

  XpuCtrl         : ST_XPU_CTRL;
  XpuState        : ST_XPU_STATE;
  XpuInfo         : ST_XPU_INFO;
  XpuModules      : ARRAY[1..MAX_MODULE] OF Tc3_XTS_Utility.ST_InfoDataView;


  //---------------------------------------------------------------------------
  // Collision avoidance group CA
  //
  // - add mover to group
  // - build group
  // - clear group
  // - whereever you may roam, no on will tread on you
  CaGroup         : FB_CaGroup;                   // cyclic check of CaGroup state and errors; carries methods for handling CaGroup
  CaGroupItf      : I_XtsTransport_CaGroup;       // Interface used by fb_TransportUnit

  // cyclic mapping to MOTION/Objects/CaGroup 
  CaGroupRef      : Tc3_McCoordinatedMotion.AXES_GROUP_REF;

  // Info data from CaGroup FB
  CaGroupInfo     : ST_GROUP_INFO;                // cyclic info about CaGroup for fb_TransportUnit to read
  //---------------------------------------------------------------------------

  //---------------------------------------------------------------------------
  // MC2 encapsulation, CA movement
  Mover                 : ARRAY[1..MAX_MOVER] OF fb_MoverCtrl;    // MC and CA methods for mover; cyclic check for individual command on mover

  MoverCtrl             : ARRAY[1..MAX_MOVER] OF ST_MOVER_CTRL;   // control of individual mover for extern to write
  MoverState            : ARRAY[1..MAX_MOVER] OF ST_MOVER_STATE;  // state   of individual mover for extern to read

  MoverSelector         : fb_MoverSelector;                       // alternative for moving a single mover via Index/ID selection
  MoverSelectorCtrl     : ST_MOVER_SELECTOR_CTRL;
  MoverSelectorState    : ST_MOVER_SELECTOR_STATE;

  MoverItf        : ARRAY[1..MAX_MOVER] OF I_XtsTransport_Mover;  // Interface used by fb_TransportUnit

  LastPosition    : ARRAY[1..MAX_MOVER] OF LREAL;           // on execute of any movement, value is saved here (used by fb_Mover)
  LastGap         : ARRAY[1..MAX_MOVER] OF LREAL;           // on execute of any movement, value is saved here (used by fb_Mover)

  MoverInfo       : ARRAY[1..MAX_MOVER] OF ST_MOVER_INFO;   // cyclic info about mover for extern to read

  MoveData        : ARRAY[1..MAX_MOVER] OF ST_MOVE_DATA;    // dynamic constraints for move commands
  GearData        : ARRAY[1..MAX_MOVER] OF ST_GEAR_DATA;    // dynamic constraints and positions for GearIn/GearInPosCa

  
  // cyclic mapping to MOTION/Axes
  AxisRefMover    : ARRAY[1..MAX_MOVER] OF Tc2_MC2.AXIS_REF;
  //---------------------------------------------------------------------------
END_VAR

// ---- XTS_TRANSPORT/GVL_XTS_VERSION.TcGVL
{attribute 'qualified_only'}
VAR_GLOBAL CONSTANT
//-----------------------------------------------------------------------------------
//-----------------------------------------------------------------------------------
// HAUD 2026 07 26
//
//    XTS_TRANSPORT_LAYER project
//    
//    MIT License
//    
//    Copyright (c) 2025 HAUD
//    
//    Permission is hereby granted, free of charge, to any person obtaining a copy
//    of this software and associated documentation files (the "Software"), to deal
//    in the Software without restriction, including without limitation the rights
//    to use, copy, modify, merge, publish, distribute, sublicense, and/or sell
//    copies of the Software, and to permit persons to whom the Software is
//    furnished to do so, subject to the following conditions:
//    
//    The above copyright notice and this permission notice shall be included in all
//    copies or substantial portions of the Software.
//    
//    THE SOFTWARE IS PROVIDED "AS IS", WITHOUT WARRANTY OF ANY KIND, EXPRESS OR
//    IMPLIED, INCLUDING BUT NOT LIMITED TO THE WARRANTIES OF MERCHANTABILITY,
//    FITNESS FOR A PARTICULAR PURPOSE AND NONINFRINGEMENT. IN NO EVENT SHALL THE
//    AUTHORS OR COPYRIGHT HOLDERS BE LIABLE FOR ANY CLAIM, DAMAGES OR OTHER
//    LIABILITY, WHETHER IN AN ACTION OF CONTRACT, TORT OR OTHERWISE, ARISING FROM,
//    OUT OF OR IN CONNECTION WITH THE SOFTWARE OR THE USE OR OTHER DEALINGS IN THE
//    SOFTWARE.
//-----------------------------------------------------------------------------------
  Version             : STRING  := '4.02.18';
//-----------------------------------------------------------------------------------
END_VAR

// ---- APPLICATION/_types/Collector/I_ProcessCollector.TcIO
INTERFACE I_ProcessCollector

PROPERTY ActivateStation : DWORD // bit mask for enabling XtsStations in Process
GET
END_GET
END_PROPERTY

METHOD PUBLIC BitDel : T_PROCESS
VAR_INPUT
  inVal   : T_PROCESS;
  bitNo   : DINT;
END_VAR
END_METHOD

METHOD PUBLIC BitGet : BOOL
VAR_INPUT
  inVal   : T_PROCESS;
  bitNo   : DINT;
END_VAR
END_METHOD

METHOD PUBLIC BitSet : T_PROCESS
VAR_INPUT
  inVal   : T_PROCESS;
  bitNo   : DINT;
END_VAR
END_METHOD

METHOD BitsToString : STRING(SIZEOF(T_PROCESS)*8) // T_PROCESS to string
VAR_INPUT
  inVal       : T_PROCESS;
END_VAR
END_METHOD

METHOD Cycle // cyclic call for checking XtsStation state masks and command input from process
END_METHOD

METHOD GetMoverInStation : ST_MOVER_INFO // mover in station info
VAR_INPUT
  nStation            : UINT;   // index of GVL_XTS.StationState[nStation]
END_VAR
END_METHOD

METHOD GetStationState : ST_STATION_STATE
VAR_INPUT
  nStation            : UINT;   // index of GVL_XTS.StationState[nStation]
END_VAR
END_METHOD

METHOD PUBLIC Init : E_PROGRESS // clears all XtsSubstations, then disables all
VAR_INPUT
  Execute     : BOOL;
END_VAR
END_METHOD

PROPERTY MessageLevel : e_MessageType
GET
END_GET
SET
END_SET
END_PROPERTY

PROPERTY ProcessCtrl : reference to st_process_ctrl
GET
END_GET
SET
END_SET
END_PROPERTY

PROPERTY ProcessId : E_INSTANCE
GET
END_GET
SET
END_SET
END_PROPERTY

PROPERTY ProcessState : reference to st_process_state
GET
END_GET
SET
END_SET
END_PROPERTY

PROPERTY QueueMoverIDs : ARRAY[1..SIZEOF(T_PROCESS)*8] OF UINT
GET
END_GET
END_PROPERTY

PROPERTY QueueProcessCount : UINT // sum of all station queues
GET
END_GET
END_PROPERTY

PROPERTY QueueStationCount : ARRAY[1..SIZEOF(T_PROCESS)*8] OF UINT
GET
END_GET
END_PROPERTY

PROPERTY StationCount : UINT
GET
END_GET
END_PROPERTY

PROPERTY StationFirst : uint
GET
END_GET
SET
END_SET
END_PROPERTY

PROPERTY StationLast : uint
GET
END_GET
SET
END_SET
END_PROPERTY

PROPERTY TargetIndex : ARRAY[1..SIZEOF(T_PROCESS)*8] OF USINT
GET
END_GET
SET
END_SET
END_PROPERTY

PROPERTY TargetMask : ARRAY[1..SIZEOF(T_PROCESS)*8] OF BYTE
GET
END_GET
SET
END_SET
END_PROPERTY

METHOD To_T_Process : T_PROCESS // maps (2^nExp)-1 onto T_PROCESS datatype 
VAR_INPUT
  nExp              : BYTE;
END_VAR
END_METHOD

END_INTERFACE

// ---- APPLICATION/_types/LinkedList/I_Process_LinkedList.TcIO
INTERFACE I_Process_LinkedList

METHOD AddHeadValue : ST_PROCESS_LIST_RESULT
VAR_INPUT
  stData        : ST_PROCESS_DATA;
END_VAR
END_METHOD

METHOD AddTailValue : ST_PROCESS_LIST_RESULT
VAR_INPUT
  stData        : ST_PROCESS_DATA;
END_VAR
END_METHOD

PROPERTY Count : UDINT
GET
END_GET
END_PROPERTY

PROPERTY Data : ARRAY[1..MAX_LIST_NODES] OF ST_PROCESS_DATA
GET
END_GET
END_PROPERTY

PROPERTY Free : UDINT
GET
END_GET
END_PROPERTY

METHOD GetHead : ST_PROCESS_LIST_RESULT
VAR_INPUT
END_VAR
END_METHOD

METHOD GetTail : ST_PROCESS_LIST_RESULT
VAR_INPUT
END_VAR
VAR
END_VAR
END_METHOD

METHOD InitList : BOOL
END_METHOD

PROPERTY Nodes : ARRAY[0..MAX_LIST_NODES] OF T_LinkedListEntry
GET
END_GET
END_PROPERTY

METHOD RemoveHeadValue : ST_PROCESS_LIST_RESULT
VAR_INPUT
END_VAR
END_METHOD

METHOD RemoveTailValue : ST_PROCESS_LIST_RESULT
VAR_INPUT
END_VAR
VAR
END_VAR
END_METHOD

END_INTERFACE

// ---- _MSG/I_MessageData.TcIO
INTERFACE I_MessageData

PROPERTY DirRoot : POINTER to string(255)
SET
END_SET
END_PROPERTY

PROPERTY ErrorIndex : reference to uint
SET
END_SET
END_PROPERTY

PROPERTY FileRoot : pointer to string(255)
SET
END_SET
END_PROPERTY

PROPERTY LocalTime : pointer to DT
SET
END_SET
END_PROPERTY

PROPERTY MessageIndex : reference to uint
SET
END_SET
END_PROPERTY

PROPERTY MsgList : pointer to ARRAY[1..GVL_MSG_XTS.MAX_MESSAGE] OF st_message
SET
END_SET
END_PROPERTY

END_INTERFACE

// ---- _XML/Configuration/I_Configuration_Station.TcIO
INTERFACE I_Configuration_Station

METHOD Check : BOOL
END_METHOD

METHOD PRIVATE Cmd : E_DATA_STATE
VAR_INPUT
  Ctrl      : E_DATA_CTRL;
END_VAR
END_METHOD

PROPERTY Ctrl : REFERENCE to ST_DATA_CTRL
SET
END_SET
END_PROPERTY

PROPERTY Identity : OTCID
GET
END_GET
SET
END_SET
END_PROPERTY

PROPERTY State : REFERENCE TO ST_DATA_STATE
SET
END_SET
END_PROPERTY

PROPERTY StationParameter : pointer to ARRAY[1..MAX_STATION] OF ST_STATION_PARAMETER
SET
END_SET
END_PROPERTY

END_INTERFACE

// ---- XTS_TRANSPORT/CaGroup/I_XtsTransport_CaGroup.TcIO
INTERFACE I_XtsTransport_CaGroup

METHOD AddAll : E_PROGRESS
VAR_INPUT
  Execute     : BOOL;
END_VAR
END_METHOD

METHOD Disable : E_PROGRESS
VAR_INPUT
  Execute     : BOOL;
END_VAR
END_METHOD

METHOD Enable : E_PROGRESS
VAR_INPUT
  Execute     : BOOL;
END_VAR
END_METHOD

METHOD McHaltAll : E_PROGRESS
VAR_INPUT
  Execute       : BOOL;
END_VAR
END_METHOD

METHOD McResetAll : E_PROGRESS
VAR_INPUT
  Execute       : BOOL;
END_VAR
END_METHOD

METHOD RemoveAll : E_PROGRESS
VAR_INPUT
  Execute     : BOOL;
END_VAR
END_METHOD

METHOD Reset : E_PROGRESS
VAR_INPUT
  Execute     : BOOL;
END_VAR
END_METHOD

METHOD Stop : E_PROGRESS
VAR_INPUT
  Execute     : BOOL;
END_VAR
END_METHOD

END_INTERFACE

// ---- XTS_TRANSPORT/Mover/I_XtsTransport_Mover.TcIO
INTERFACE I_XtsTransport_Mover

METHOD Disable : E_PROGRESS
VAR_INPUT
  Execute             : BOOL;
END_VAR
END_METHOD

METHOD Enable : E_PROGRESS
VAR_INPUT
  Execute             : BOOL;
END_VAR
END_METHOD

METHOD GearIn : E_PROGRESS;
VAR_INPUT
  Execute             : BOOL;
  stMoveData          : ST_MOVE_DATA;
  stGearData          : ST_GEAR_DATA;
END_VAR
END_METHOD

METHOD GearInPosCa : E_PROGRESS
VAR_INPUT
  Execute             : BOOL;
  stMoveData          : ST_MOVE_DATA;
  stGearData          : ST_GEAR_DATA;  
END_VAR
END_METHOD

METHOD GearOut : E_PROGRESS
VAR_INPUT
  Execute             : BOOL;
END_VAR
END_METHOD

METHOD Halt : E_PROGRESS
VAR_INPUT
  Execute             : BOOL;
  stMoveData          : ST_MOVE_DATA;
END_VAR
END_METHOD

METHOD HaltCa : E_PROGRESS
VAR_INPUT
  Execute             : BOOL;
  stMoveData          : ST_MOVE_DATA;
END_VAR
END_METHOD

PROPERTY Master : REFERENCE to AXIS_REF
SET
END_SET
END_PROPERTY

PROPERTY MessageLevel : e_messagetype
SET
END_SET
END_PROPERTY

PROPERTY ModuloTurn : dint
GET
END_GET
END_PROPERTY

METHOD MoveToPos : E_PROGRESS
VAR_INPUT
  Execute             : BOOL;
  stMoveData          : ST_MOVE_DATA;
END_VAR
END_METHOD

METHOD MoveToPosCa : E_PROGRESS
VAR_INPUT
  Execute             : BOOL;
  stMoveData          : ST_MOVE_DATA;
END_VAR
END_METHOD

PROPERTY RailLength : LREAL
GET
END_GET
SET
END_SET
END_PROPERTY

METHOD Reset : E_PROGRESS
VAR_INPUT
  Execute             : BOOL;
END_VAR
END_METHOD

METHOD SendToAbsPosCa : E_PROGRESS
VAR_INPUT
  Execute             : BOOL;
  stMoveData          : ST_MOVE_DATA;
END_VAR
END_METHOD

METHOD SendToModuloPosCa : E_PROGRESS
VAR_INPUT
  Execute             : BOOL;
  stMoveData          : ST_MOVE_DATA;
END_VAR
END_METHOD

METHOD Stop : E_PROGRESS
VAR_INPUT
  Execute             : BOOL;
  stMoveData          : ST_MOVE_DATA;
END_VAR
END_METHOD

END_INTERFACE

// ---- XTS_TRANSPORT/Xpu/I_XtsTransport_Xpu.TcIO
INTERFACE I_XtsTransport_Xpu

METHOD GetEnvironment : I_TcIoXtsEnvironment
VAR_INPUT
END_VAR
END_METHOD

METHOD GetNctBaseUnit : Tc3_XTS_Utility.I_TcIoXtsNctBaseUnitInterface
VAR_INPUT
  Index     : UINT;
END_VAR
END_METHOD

METHOD GetNctController : Tc3_XTS_Utility.I_TcIoXtsNctController
VAR_INPUT
END_VAR
END_METHOD

METHOD GetParameterSet : I_TcIoXtsParameterSet
VAR_INPUT
  Index     : UINT;
END_VAR
END_METHOD

METHOD GetPartModules : ARRAY[1..MAX_MODULE]  OF Tc3_XTS_Utility.I_TcIoXtsPartModule;
VAR_INPUT
END_VAR
END_METHOD

METHOD GetProcessingUnit : Tc3_XTS_Utility.I_TcIoXtsProcessingUnit
VAR_INPUT
END_VAR
END_METHOD

END_INTERFACE

// ---- XTS_TRANSPORT/XtsStation/I_XtsTransport_Station.TcIO
INTERFACE I_XtsTransport_Station

METHOD Init : e_progress
VAR_INPUT
END_VAR
END_METHOD

PROPERTY MessageLevel : e_messagetype
SET
END_SET
END_PROPERTY

PROPERTY StationId : uint // know thy reflection,
GET
END_GET
SET
END_SET
END_PROPERTY

PROPERTY TargetWindow : lreal
GET
END_GET
SET
END_SET
END_PROPERTY

END_INTERFACE

// ---- XTS_TRANSPORT/XtsStation/types/I_Station_LinkedList.TcIO
INTERFACE I_Station_LinkedList

METHOD AddHeadValue : ST_STATION_LIST_RESULT
VAR_INPUT
  stData        : ST_STATION_MOVER_DATA;
END_VAR
END_METHOD

METHOD AddTailValue : ST_STATION_LIST_RESULT
VAR_INPUT
  stData          : ST_STATION_MOVER_DATA;
END_VAR
END_METHOD

PROPERTY Count : UDINT
GET
END_GET
END_PROPERTY

PROPERTY Data : ARRAY[1..MAX_LIST_NODES] OF ST_STATION_MOVER_DATA
GET
END_GET
END_PROPERTY

PROPERTY Free : UDINT
GET
END_GET
END_PROPERTY

METHOD GetHead : ST_STATION_LIST_RESULT
VAR_INPUT
END_VAR
END_METHOD

METHOD InitList : BOOL
END_METHOD

PROPERTY Nodes : ARRAY[0..MAX_LIST_NODES] OF T_LinkedListEntry
GET
END_GET
END_PROPERTY

METHOD RemoveHeadValue : ST_STATION_LIST_RESULT
VAR_INPUT
END_VAR
END_METHOD

END_INTERFACE

// ---- MAPPING/MAPPING_XTS_in.TcPOU
PROGRAM MAPPING_XTS_in
//-----------------------------------------------------------------------------------------------------------------
//
//  HAUD 2026.02.24
//
//  - MAPPING : "It's not the best choice, it's the only choice!" 
//
//    - Spacer's Choice: barrier of entry
//      - memcpy? --> This is the law.
//
//      - everyone coming in from any other cyclic realm has to pass this border
//      - instatiates control structures at compile
//      - use of compiler defines
//      - cyclic validation for matching sizes
//-----------------------------------------------------------------------------------------------------------------
VAR CONSTANT
//-----------------------------------------------------------------------------------------------------------------
//  - compiler defines check
//    - you find the compiler defines in the plc project properties under section Compile
//-----------------------------------------------------------------------------------------------------------------
{IF defined (MOVER_MAP)}
  {info 'XTS_TRANSPORT_LAYER: - MOVER_MAPPING active'}
  bBypassMappingMover       : BOOL  := FALSE;
  bMoverSelector            : BOOL  := FALSE;
{ELSE}
  // HAUD 2026 04 20
  // - selector is now configurable via compile
  {IF defined (MOVER_SELECTOR)}
    {info 'XTS_TRANSPORT_LAYER: - MOVER_SELECTOR active'}
    bBypassMappingMover     : BOOL  := FALSE;
    bMoverSelector          : BOOL  := TRUE;
  {ELSE}
    bBypassMappingMover     : BOOL  := TRUE;
    bMoverSelector          : BOOL  := FALSE;
  {END_IF}
{END_IF}
//-----------------------------------------------------------------------------------------------------------------
//-----------------------------------------------------------------------------------------------------------------
{IF defined (STATION_MAP)}
  {info 'XTS_TRANSPORT_LAYER: - STATION_MAPPING active'}
  bBypassMappingStation     : BOOL  := FALSE;
{ELSE}
  bBypassMappingStation     : BOOL  := TRUE;
{END_IF}
END_VAR
VAR
//-----------------------------------------------------------------------------------------------------------------
//  - bypass and state info
//-----------------------------------------------------------------------------------------------------------------
  bBypass                   : BOOL    := TRUE;  // local switch for local control
  sMappingCheck             : STRING;           // Work invigorates the spirit.
//-----------------------------------------------------------------------------------------------------------------
//  - compiler defines check
//-----------------------------------------------------------------------------------------------------------------
{IF defined (MOVER_MAP)}
  MoverCtrl                 : U_MOVER_CTRL;     // individual mover control
  MoveData                  : U_MOVE_DATA;      // parameter set for movements
  GearData                  : U_GEAR_DATA;      // additional parameter set for geared in motion
{ELSE}
  // HAUD 2026 04 20
  // - selector is now configurable via compile
  {IF defined (MOVER_SELECTOR)}
    MoverCtrl               : U_MOVER_SELECTOR_CTRL;  // SELECTIVE mover control
    MoveData                : U_MOVE_DATA;            // parameter set for movement
    GearData                : U_GEAR_DATA;            // additional parameter set for geared in motion
  {ELSE}
    MoverCtrl               : BYTE;
    MoveData                : BYTE;
    GearData                : BYTE;
  {END_IF}
{END_IF}
//-----------------------------------------------------------------------------------------------------------------
//-----------------------------------------------------------------------------------------------------------------
{IF defined (STATION_MAP)}
  StationControl            : U_XTS_STATION_CTRL;   // traffic control
{ELSE}
  StationControl            : BYTE;
{END_IF}
//-----------------------------------------------------------------------------------------------------------------
//-----------------------------------------------------------------------------------------------------------------
{IF (defined (STATION_MAP)) OR (defined (MOVER_MAP)) OR (defined(MOVER_SELECTOR))}
  {info 'XTS_TRANSPORT_LAYER: - TransportControl'}
  TransportControl          : U_XTS_TRANSPORT_CTRL; // UDL-001 the Groundbreaker
{ELSE}
  TransportControl          : BYTE;
{END_IF}
//-----------------------------------------------------------------------------------------------------------------
//  - size checks
//-----------------------------------------------------------------------------------------------------------------
  szGearData,
  szMoveData,
  szMoverCtrl               : ARRAY[1..2] OF UDINT;

  szStationCtrl             : ARRAY[1..2] OF UDINT;

  szTransportCtrl           : ARRAY[1..2] OF UDINT;
//-----------------------------------------------------------------------------------------------------------------
//  - destination poiners
//-----------------------------------------------------------------------------------------------------------------
  pMoverCtrl                : pvoid;
  pMoveData                 : pvoid;
  pGearData                 : pvoid;
END_VAR

//--------------------------------------------------------------------------------------------
//  - datafield size check
//--------------------------------------------------------------------------------------------
IF NOT Check() THEN RETURN; END_IF
//--------------------------------------------------------------------------------------------
//--------------------------------------------------------------------------------------------
//--------------------------------------------------------------------------------------------
//  - bypass switch
//--------------------------------------------------------------------------------------------
IF (bBypass) 
THEN 
  sMappingCheck  := 'BYPASS_SWITCHED_ON';
  RETURN;
END_IF
//--------------------------------------------------------------------------------------------
//--------------------------------------------------------------------------------------------
//           destination,                   source,                    size
//--------------------------------------------------------------------------------------------
IF NOT bBypassMappingMover
THEN
  IF NOT bMoverSelector
  THEN
    pMoverCtrl    := ADR(GVL_XTS.MoverCtrl);
    pMoveData     := ADR(GVL_XTS.MoveData);
    pGearData     := ADR(GVL_XTS.GearData);
  ELSE
    pMoverCtrl    := ADR(GVL_XTS.MoverSelectorCtrl);
    pMoveData     := ADR(GVL_XTS.MoveData);
    pGearData     := ADR(GVL_XTS.GearData);
  END_IF

  memcpy(pMoverCtrl,                    ADR(MoverCtrl),         SIZEOF(MoverCtrl));
  memcpy(pMoveData ,                    ADR(MoveData) ,         SIZEOF(MoveData));
  memcpy(pGearData ,                    ADR(GearData) ,         SIZEOF(GearData));
END_IF
//--------------------------------------------------------------------------------------------
//--------------------------------------------------------------------------------------------
IF NOT bBypassMappingStation
THEN
  memcpy(ADR(GVL_XTS.StationCtrl),      ADR(StationControl),    SIZEOF(StationControl));
END_IF
//--------------------------------------------------------------------------------------------
//--------------------------------------------------------------------------------------------
IF NOT bBypassMappingStation OR
   NOT bBypassMappingMover
THEN
  memcpy(ADR(GVL_XTS.XtsTransportCtrl), ADR(TransportControl),  SIZEOF(TransportControl));
END_IF
//--------------------------------------------------------------------------------------------
//           destination,                   source,                    size
//--------------------------------------------------------------------------------------------
//--------------------------------------------------------------------------------------------

PROPERTY BypassSwitch : BOOL
GET
BypassSwitch := bBypass;
END_GET
SET
bBypass := BypassSwitch;
END_SET
END_PROPERTY

